// TwinCAT 3 PLC project MasterController
// ProgramVersion: 3.1.4024.0
// libraries:
//   Tc2_EtherCAT, * (Beckhoff Automation GmbH)
//   Tc2_Math, * (Beckhoff Automation GmbH)
//   Tc2_Standard, * (Beckhoff Automation GmbH)
//   Tc2_System, * (Beckhoff Automation GmbH)
//   Tc2_Utilities, * (Beckhoff Automation GmbH)
//   Tc3_Module, * (Beckhoff Automation GmbH)
// project tree:
//   AgiMaths/Frames/ DHTrans.TcPOU (not stored), invFrame.TcPOU (not stored), rotX.TcPOU (not stored), rotY.TcPOU (not stored), rotZ.TcPOU (not stored), transform.TcPOU (not stored)
//   AgiMaths/MatrixLib/ angAxis2Rot.TcPOU (not stored), cross.TcPOU (not stored), Det5.TcPOU (not stored), Det6.TcPOU (not stored), Det7.TcPOU (not stored), invMat6.TcPOU (not stored), invMat6Old.TcPOU (not stored), invMat3.TcPOU (not stored), invMat7.TcPOU (not stored), Mat3T.TcPOU (not stored), matAdd.TcPOU (not stored), matMultiNum.TcPOU (not stored), matMultiply.TcPOU (not stored), matMultiVec.TcPOU (not stored), matSelfAdd.TcPOU (not stored), matSelfSub.TcPOU (not stored), matSub.TcPOU (not stored), matTranspose.TcPOU (not stored), rot2AngAxis.TcPOU (not stored), norm.TcPOU (not stored), normalize.TcPOU (not stored), vecAdd.TcPOU (not stored), vecDot.TcPOU (not stored), vecMultiNum.TcPOU (not stored), vecSelfAdd.TcPOU (not stored), vecSelfMultiNum.TcPOU (not stored), vecSelfSub.TcPOU (not stored), vecSub.TcPOU (not stored)
//   AgiMaths/ sign.TcPOU (not stored), addVec7.TcPOU (not stored), atan2.TcPOU (not stored), cot.TcPOU (not stored)
//   DUTs/Enum/ E_InstruEnergyCtrlWord.TcDUT (not stored), E_InstrumentEnergyType.TcDUT (not stored), E_InstrumentType.TcDUT (not stored), E_MasterArmState.TcDUT (not stored), E_MatchedSlaveArmIdx.TcDUT (not stored), E_SlaveArmState.TcDUT (not stored), E_DriverCtrlWord.TcDUT (not stored), E_DriverOPMode.TcDUT (not stored), E_DriverStatusWord.TcDUT (not stored)
//   DUTs/Structure/MasterSlaveCommunication/ ST_MasterStatus.TcDUT (not stored), ST_SlaveStatus.TcDUT (not stored)
//   DUTs/Structure/ ST_EtherCATState.TcDUT (not stored), ST_InstruStatus.TcDUT (not stored), ST_MatchedMasterArmIdx.TcDUT (not stored), ST_ArmCtrlCmds.TcDUT (not stored), ST_MasterInputDataPool.TcDUT (not stored), ST_Frame.TcDUT (not stored)
//   DUTs/Structure/TasksCommunication/ ST_CartUIData.TcDUT (not stored), ST_MasterDynaData.TcDUT (not stored), ST_MasterUIData.TcDUT (not stored), ST_CartStatus.TcDUT (not stored), ST_MasterJointData.TcDUT (not stored), ST_MotorInputs.TcDUT (not stored), ST_MotorOutputs.TcDUT (not stored), ST_SlaveJointData.TcDUT (not stored), ST_SafetyData.TcDUT (not stored), ST_CartJointData.TcDUT (not stored)
//   DUTs/Structure/UICommunication/ ST_arm_distribution.TcDUT (not stored), ST_ergonCtrlEnable.TcDUT (not stored), ST_ergonomicCtrlData.TcDUT (not stored), ST_instrument_info.TcDUT (not stored), ST_scope_info.TcDUT (not stored)
//   DUTs/Type/ Vec7b.TcDUT (not stored), Mat34.TcDUT (not stored), Mat37.TcDUT (not stored), Mat43.TcDUT (not stored), Mat4d.TcDUT (not stored), Mat5d.TcDUT (not stored), Mat67.TcDUT (not stored), Mat6d.TcDUT (not stored), Mat76.TcDUT (not stored), Mat7d.TcDUT (not stored), Vec4d.TcDUT (not stored), Vec4i.TcDUT (not stored), Vec6i.TcDUT (not stored), Vec4b.TcDUT (not stored), Vec7di.TcDUT (not stored), Vec8d.TcDUT (not stored), Mat3d.TcDUT (not stored), Vec3d.TcDUT (not stored), Vec6d.TcDUT (not stored), Vec7d.TcDUT (not stored), Vec7i.TcDUT (not stored)
//   FBs_Auxiliary/ FB_GripAngleCalc.TcPOU, FB_HandClutchCheck.TcPOU (not stored), FB_IOCheck.TcPOU (not stored), FB_RiseEdgeCheck.TcPOU (not stored), FB_IOToggleCheck.TcPOU (not stored), FB_MSCtrlTriggerCheck.TcPOU (not stored), FB_slaveConnectionCheck.TcPOU (not stored), FB_TON.TcPOU (not stored)
//   FBs_BasicControllers/ FB_boundaryForceFeedback.TcPOU (not stored), FB_Jnt6SWLimit.TcPOU (not stored), FB_PID.TcPOU (not stored), FB_RedunJntControl.TcPOU (not stored)
//   FBs_Observer/ FB_JntObserver.TcPOU (not stored)
//   FBs_RobotDynamics/ FB_MasterDynamic.TcPOU (not stored), FB_MasterFriciton.TcPOU (not stored), FB_MasterGravity.TcPOU (not stored)
//   FBs_Robots/ FB_ArmJoint.TcPOU (not stored), FB_CartJoint.TcPOU, FB_JointBase.TcPOU, FB_MasterCart.TcPOU, FB_MasterArm.TcPOU (not stored), FB_MasterRobot.TcPOU
//   FBs_StateControllers/ FB_EndoscopeController.TcPOU (not stored), FB_StateCtrlClutch.TcPOU (not stored), FB_StateCtrlEndoscope.TcPOU (not stored), FB_StateCtrlCart.TcPOU (not stored), FB_StateCtrlDisable.TcPOU (not stored), FB_StateCtrlGraCali.TcPOU (not stored), FB_StateCtrlMatching.TcPOU, FB_StateCtrlHome.TcPOU (not stored), FB_StateCtrlError.TcPOU (not stored), FB_StateCtrlPerformance.TcPOU (not stored), FB_StateCtrlReady.TcPOU (not stored), FB_StateCtrlMasterSlave.TcPOU (not stored), FB_StateCtrlTest.TcPOU (not stored), FB_StateCtrlInit.TcPOU (not stored), FB_StateCtrlStandBy.TcPOU (not stored), FB_MasterArmCtrlBase.TcPOU (not stored), I_MasterArmCtrl.TcIO (not stored)
//   FBs_TrajectoryPlanning/ FB_BasicDoubleS.TcPOU (not stored), FB_trajBase.TcPOU (not stored), FB_TrajMoveJ.TcPOU (not stored), linear_trajectory_with_quintic_polynomial_blends.TcPOU (not stored), quintic_spline_curve.TcPOU (not stored), Quintic_spline_curve_factor.TcPOU (not stored), TrapezoIDal_velocity_trajectory.TcPOU (not stored)
//   FBs_TrajectoryPlanning/OTG/ FB_secOrdTrajFilter.TcPOU (not stored), FB_thirdOrdTrajFilter.TcPOU (not stored)
//   FBs_Filters/ FB_LowPassFilter.TcPOU (not stored)
//   GVLs/Arms/ GVL_ArmDynamics.TcGVL, GVL_ArmJointCaliData.TcGVL, GVL_ArmKinematic.TcGVL, GVL_ControlParameters.TcGVL (not stored), GVL_ArmJointParameters.TcGVL (not stored)
//   GVLs/Cart/ GVL_CartJointCaliData.TcGVL (not stored), GVL_CartJointParameters.TcGVL (not stored)
//   GVLs/Configs/Robot3/ GVL_ArmDynamics_3.TcGVL (not stored), GVL_ArmJointCaliData_3.TcGVL (not stored), GVL_CartJointCaliData_3.TcGVL (not stored)
//   GVLs/Configs/Robot4/ GVL_ArmDynamics_4.TcGVL (not stored), GVL_ArmJointCaliData_4.TcGVL (not stored), GVL_CartJointCaliData_4_1.TcGVL (not stored)
//   GVLs/Configs/Robot5/ GVL_ArmDynamics_5.TcGVL (not stored), GVL_ArmJointCaliData_5.TcGVL (not stored), GVL_CartJointCaliData_5.TcGVL (not stored)
//   GVLs/Configs/Robot6/ GVL_ArmDynamics_6.TcGVL (not stored), GVL_ArmJointCaliData_6.TcGVL (not stored), GVL_CartJointCaliData_6.TcGVL (not stored)
//   GVLs/ GVL_interactUI.TcGVL (not stored), GVL_MathDefine.TcGVL (not stored), GVL_SafetyParameters.TcGVL, GVL_SystemParameters.TcGVL (not stored)
//   Mains/ CartControl.TcPOU (not stored), SafetyCheck.TcPOU (not stored), MasterArmControl.TcPOU (not stored), RobotDynamics.TcPOU (not stored)
//   SafetyCheck/ ASSERT.TcPOU (not stored), Fb_dataRecord.TcPOU (not stored), FB_EtherCATCheck.TcPOU (not stored), Fb_SafetyCheck.TcPOU, FB_Writer.TcPOU (not stored)
//   SafetyCheck/safetyCheckDUT/ checkDelay.TcDUT (not stored), checkDelayTime.TcDUT (not stored), checkInputVariable.TcDUT (not stored), checkPermit.TcDUT (not stored), ST_Buffer.TcDUT (not stored), T_Buffer.TcDUT (not stored)
//   Sandbox/ FB_CartCheck.TcPOU (not stored), FB_MasterArmCheck.TcPOU (not stored), FB_RedunJntControl_bak2.TcPOU (not stored), FB_RedunJntControl_bak.TcPOU (not stored)
//   / TaskArmControl.TcTTO (not stored), TaskCartControl.TcTTO (not stored), TaskDynamic.TcTTO (not stored), TaskSafetyCheck.TcTTO (not stored)
// real-time tasks:
//   TASK TaskArmControl: cycle T#250us, priority 1, ADS port 350
//   TASK TaskDynamic: cycle T#1ms, priority 2, ADS port 351
//   TASK TaskSafetyCheck: cycle T#1ms, priority 5, ADS port 352
//   TASK TaskCartControl: cycle T#1ms, priority 4, ADS port 353
// I/O:
//   DEVICE RightArm (EtherCAT), AmsNetId 169.254.219.236.5.1
//     Term 7 (EK1100) [EK1100 EtherCAT Coupler (2A E-Bus)]
//       Term 8 (EL6070) [EL6070 1Ch. Licensing-Terminal]
//       Term 9 (EL1008) [EL1008 8Ch. Dig. Input 24V, 3ms]
//       Term 10 (EL1008) [EL1008 8Ch. Dig. Input 24V, 3ms]
//       Term 11 (EL1008) [EL1008 8Ch. Dig. Input 24V, 3ms]
//       Term 12 (EK1122) [EK1122 2 port EtherCAT junction]
//         Box 13 (AX58200_MotorControl) [AX58200_MotorControl_for_1axis]
//         Box 14 (AX58200_MotorControl) [AX58200_MotorControl_for_1axis]
//         Box 15 (AX58200_MotorControl) [AX58200_MotorControl_for_1axis]
//         Box 16 (AX58200_MotorControl) [AX58200_MotorControl_for_1axis]
//     Joint12 [AX58200_MotorControl_Master123]
//     Joint3 [AX58200_MotorControl_Master123]
//     Joint4 [AX58200_MotorControl_for_1axis]
//     Joint5 [AX58200_MotorControl_for_1axis]
//     Joint6 [AX58200_MotorControl_for_1axis]
//     Joint7 [AX58200_MotorControl_for_1axis]
//   DEVICE LeftArm (EtherCAT), AmsNetId 169.254.79.95.2.1
//     Joint12 [AX58200_MotorControl_Master123]
//     Joint3 [AX58200_MotorControl_Master123]
//     Joint4 [AX58200_MotorControl_for_1axis]
//     Joint5 [AX58200_MotorControl_for_1axis]
//     Joint6 [AX58200_MotorControl_for_1axis]
//     Joint7 [AX58200_MotorControl_for_1axis]
//   DEVICE Device 3 (EtherCAT), AmsNetId 169.254.219.236.4.1
//     Box 2 (AX58200_MotorControl) [AX58200_MotorControlHFK]
//     Box 1 (EL6695-0002) [EL6695 EtherCAT Bridge terminal (Secondary)]
// variable links:
//   MasterController/MasterController Instance <-> Device 3 (EtherCAT)/Box 1 (EL6695-0002)
//     TaskArmControl Inputs/MasterArmControl.m_slaveRobotData <-> IO Inputs/SlaveRobotData
//     TaskArmControl Outputs/MasterArmControl.m_masterRobotData <-> IO Outputs/MasterRobotData
//   MasterController/MasterController Instance <-> Device 3 (EtherCAT)/Box 2 (AX58200_MotorControl)
//     TaskCartControl Outputs/CartControl.m_masterCart.m_elecKnifeCtrlWord <-> RxPdoMappingCspCsv/Target velocity
//   MasterController/MasterController Instance <-> LeftArm (EtherCAT)/Joint12
//     TaskArmControl Inputs/MasterArmControl.m_masterRobot.m_masterArms[1].m_joints[1].m_motorInputs/m_current <-> TxPdoMappingCspCsv/Torque actual value
//     TaskArmControl Inputs/MasterArmControl.m_masterRobot.m_masterArms[1].m_joints[1].m_motorInputs/m_driverError <-> TxPdoMappingCspCsv/digital input
//     TaskArmControl Inputs/MasterArmControl.m_masterRobot.m_masterArms[1].m_joints[2].m_motorInputs/m_driverError <-> TxPdoMappingCspCsv/digital input
//     TaskArmControl Inputs/MasterArmControl.m_masterRobot.m_masterArms[1].m_joints[1].m_motorInputs/m_motorEncoder <-> TxPdoMappingCspCsv/Position actual value
//     TaskArmControl Inputs/MasterArmControl.m_masterRobot.m_masterArms[1].m_joints[1].m_motorInputs/m_statusWord <-> TxPdoMappingCspCsv/Statusword
//     TaskArmControl Inputs/MasterArmControl.m_masterRobot.m_masterArms[1].m_joints[2].m_motorInputs/m_statusWord <-> TxPdoMappingCspCsv/Statusword
//     TaskArmControl Inputs/MasterArmControl.m_masterRobot.m_masterArms[1].m_joints[2].m_motorInputs/m_current <-> TxPdoMappingCspCsv/Torque actual value for aix2
//     TaskArmControl Inputs/MasterArmControl.m_masterRobot.m_masterArms[1].m_joints[2].m_motorInputs/m_motorEncoder <-> TxPdoMappingCspCsv/Position actual value for aix2
//     TaskArmControl Inputs/MasterArmControl.m_masterRobot.m_masterArms[1].m_joints[3].m_motorInputs/m_linkEncoder <-> TxPdoMappingCspCsv/ENC2
//     TaskArmControl Outputs/MasterArmControl.m_masterRobot.m_masterArms[1].m_joints[1].m_motorOutputs/m_cmdCurrent <-> RxPdoMappingCspCsv/Target torque
//     TaskArmControl Outputs/MasterArmControl.m_masterRobot.m_masterArms[1].m_joints[1].m_motorOutputs/m_cmdMotorEncoder <-> RxPdoMappingCspCsv/Target position
//     TaskArmControl Outputs/MasterArmControl.m_masterRobot.m_masterArms[1].m_joints[1].m_motorOutputs/m_controlWord <-> RxPdoMappingCspCsv/Controlword
//     TaskArmControl Outputs/MasterArmControl.m_masterRobot.m_masterArms[1].m_joints[1].m_motorOutputs/m_opMode <-> RxPdoMappingCspCsv/Modes of operation
//     TaskArmControl Outputs/MasterArmControl.m_masterRobot.m_masterArms[1].m_joints[2].m_motorOutputs/m_cmdCurrent <-> RxPdoMappingCspCsv/Target Torque value for aix2
//     TaskArmControl Outputs/MasterArmControl.m_masterRobot.m_masterArms[1].m_joints[2].m_motorOutputs/m_cmdMotorEncoder <-> RxPdoMappingCspCsv/Target position value for aix2
//   MasterController/MasterController Instance <-> LeftArm (EtherCAT)/Joint3
//     TaskArmControl Inputs/MasterArmControl.m_masterRobot.m_masterArms[1].m_joints[1].m_motorInputs/m_linkEncoder <-> TxPdoMappingCspCsv/ENC2
//     TaskArmControl Inputs/MasterArmControl.m_masterRobot.m_masterArms[1].m_joints[3].m_motorInputs/m_current <-> TxPdoMappingCspCsv/Torque actual value
//     TaskArmControl Inputs/MasterArmControl.m_masterRobot.m_masterArms[1].m_joints[3].m_motorInputs/m_driverError <-> TxPdoMappingCspCsv/digital input
//     TaskArmControl Inputs/MasterArmControl.m_masterRobot.m_masterArms[1].m_joints[3].m_motorInputs/m_motorEncoder <-> TxPdoMappingCspCsv/Position actual value
//     TaskArmControl Inputs/MasterArmControl.m_masterRobot.m_masterArms[1].m_joints[3].m_motorInputs/m_statusWord <-> TxPdoMappingCspCsv/Statusword
//     TaskArmControl Outputs/MasterArmControl.m_masterRobot.m_masterArms[1].m_joints[3].m_motorOutputs/m_cmdCurrent <-> RxPdoMappingCspCsv/Target torque
//     TaskArmControl Outputs/MasterArmControl.m_masterRobot.m_masterArms[1].m_joints[3].m_motorOutputs/m_cmdMotorEncoder <-> RxPdoMappingCspCsv/Target position
//     TaskArmControl Outputs/MasterArmControl.m_masterRobot.m_masterArms[1].m_joints[3].m_motorOutputs/m_controlWord <-> RxPdoMappingCspCsv/Controlword
//     TaskArmControl Outputs/MasterArmControl.m_masterRobot.m_masterArms[1].m_joints[3].m_motorOutputs/m_opMode <-> RxPdoMappingCspCsv/Modes of operation
//   MasterController/MasterController Instance <-> LeftArm (EtherCAT)/Joint4
//     TaskArmControl Inputs/MasterArmControl.m_masterRobot.m_masterArms[1].m_joints[2].m_motorInputs/m_linkEncoder <-> TxPdoMappingCspCsv/Velocity actual value
//     TaskArmControl Inputs/MasterArmControl.m_masterRobot.m_masterArms[1].m_joints[4].m_motorInputs/m_current <-> TxPdoMappingCspCsv/Torque actual value
//     TaskArmControl Inputs/MasterArmControl.m_masterRobot.m_masterArms[1].m_joints[4].m_motorInputs/m_driverError <-> TxPdoMappingCspCsv/digital input
//     TaskArmControl Inputs/MasterArmControl.m_masterRobot.m_masterArms[1].m_joints[4].m_motorInputs/m_linkEncoder <-> TxPdoMappingCspCsv/ENC2
//     TaskArmControl Inputs/MasterArmControl.m_masterRobot.m_masterArms[1].m_joints[4].m_motorInputs/m_motorEncoder <-> TxPdoMappingCspCsv/Position actual value
//     TaskArmControl Inputs/MasterArmControl.m_masterRobot.m_masterArms[1].m_joints[4].m_motorInputs/m_statusWord <-> TxPdoMappingCspCsv/Statusword
//     TaskArmControl Outputs/MasterArmControl.m_masterRobot.m_masterArms[1].m_joints[4].m_motorOutputs/m_cmdCurrent <-> RxPdoMappingCspCsv/Target torque
//     TaskArmControl Outputs/MasterArmControl.m_masterRobot.m_masterArms[1].m_joints[4].m_motorOutputs/m_cmdMotorEncoder <-> RxPdoMappingCspCsv/Target position
//     TaskArmControl Outputs/MasterArmControl.m_masterRobot.m_masterArms[1].m_joints[4].m_motorOutputs/m_controlWord <-> RxPdoMappingCspCsv/Controlword
//     TaskArmControl Outputs/MasterArmControl.m_masterRobot.m_masterArms[1].m_joints[4].m_motorOutputs/m_opMode <-> RxPdoMappingCspCsv/Modes of operation
//   MasterController/MasterController Instance <-> LeftArm (EtherCAT)/Joint5
//     TaskArmControl Inputs/MasterArmControl.m_masterRobot.m_masterArms[1].m_joints[5].m_motorInputs/m_current <-> TxPdoMappingCspCsv/Torque actual value
//     TaskArmControl Inputs/MasterArmControl.m_masterRobot.m_masterArms[1].m_joints[5].m_motorInputs/m_driverError <-> TxPdoMappingCspCsv/digital input
//     TaskArmControl Inputs/MasterArmControl.m_masterRobot.m_masterArms[1].m_joints[5].m_motorInputs/m_linkEncoder <-> TxPdoMappingCspCsv/ENC2
//     TaskArmControl Inputs/MasterArmControl.m_masterRobot.m_masterArms[1].m_joints[5].m_motorInputs/m_motorEncoder <-> TxPdoMappingCspCsv/Position actual value
//     TaskArmControl Inputs/MasterArmControl.m_masterRobot.m_masterArms[1].m_joints[5].m_motorInputs/m_statusWord <-> TxPdoMappingCspCsv/Statusword
//     TaskArmControl Outputs/MasterArmControl.m_masterRobot.m_masterArms[1].m_joints[5].m_motorOutputs/m_cmdCurrent <-> RxPdoMappingCspCsv/Target torque
//     TaskArmControl Outputs/MasterArmControl.m_masterRobot.m_masterArms[1].m_joints[5].m_motorOutputs/m_cmdMotorEncoder <-> RxPdoMappingCspCsv/Target position
//     TaskArmControl Outputs/MasterArmControl.m_masterRobot.m_masterArms[1].m_joints[5].m_motorOutputs/m_controlWord <-> RxPdoMappingCspCsv/Controlword
//     TaskArmControl Outputs/MasterArmControl.m_masterRobot.m_masterArms[1].m_joints[5].m_motorOutputs/m_opMode <-> RxPdoMappingCspCsv/Modes of operation
//   MasterController/MasterController Instance <-> LeftArm (EtherCAT)/Joint6
//     TaskArmControl Inputs/MasterArmControl.m_masterRobot.m_masterArms[1].m_joints[6].m_motorInputs/m_current <-> TxPdoMappingCspCsv/Torque actual value
//     TaskArmControl Inputs/MasterArmControl.m_masterRobot.m_masterArms[1].m_joints[6].m_motorInputs/m_driverError <-> TxPdoMappingCspCsv/digital input
//     TaskArmControl Inputs/MasterArmControl.m_masterRobot.m_masterArms[1].m_joints[6].m_motorInputs/m_linkEncoder <-> TxPdoMappingCspCsv/ENC2
//     TaskArmControl Inputs/MasterArmControl.m_masterRobot.m_masterArms[1].m_joints[6].m_motorInputs/m_motorEncoder <-> TxPdoMappingCspCsv/Position actual value
//     TaskArmControl Inputs/MasterArmControl.m_masterRobot.m_masterArms[1].m_joints[6].m_motorInputs/m_statusWord <-> TxPdoMappingCspCsv/Statusword
//     TaskArmControl Outputs/MasterArmControl.m_masterRobot.m_masterArms[1].m_joints[6].m_motorOutputs/m_cmdCurrent <-> RxPdoMappingCspCsv/Target torque
//     TaskArmControl Outputs/MasterArmControl.m_masterRobot.m_masterArms[1].m_joints[6].m_motorOutputs/m_cmdMotorEncoder <-> RxPdoMappingCspCsv/Target position
//     TaskArmControl Outputs/MasterArmControl.m_masterRobot.m_masterArms[1].m_joints[6].m_motorOutputs/m_controlWord <-> RxPdoMappingCspCsv/Controlword
//     TaskArmControl Outputs/MasterArmControl.m_masterRobot.m_masterArms[1].m_joints[6].m_motorOutputs/m_opMode <-> RxPdoMappingCspCsv/Modes of operation
//   MasterController/MasterController Instance <-> LeftArm (EtherCAT)/Joint7
//     TaskArmControl Inputs/MasterArmControl.m_masterRobot.m_masterArms[1].m_gripHallSensorIO <-> TxPdoMappingCspCsv/analog input
//     TaskArmControl Inputs/MasterArmControl.m_masterRobot.m_masterArms[1].m_handClutchIO <-> TxPdoMappingCspCsv/digital input
//     TaskArmControl Inputs/MasterArmControl.m_masterRobot.m_masterArms[1].m_joints[7].m_motorInputs/m_current <-> TxPdoMappingCspCsv/Torque actual value
//     TaskArmControl Inputs/MasterArmControl.m_masterRobot.m_masterArms[1].m_joints[7].m_motorInputs/m_linkEncoder <-> TxPdoMappingCspCsv/ENC2
//     TaskArmControl Inputs/MasterArmControl.m_masterRobot.m_masterArms[1].m_joints[7].m_motorInputs/m_motorEncoder <-> TxPdoMappingCspCsv/Position actual value
//     TaskArmControl Inputs/MasterArmControl.m_masterRobot.m_masterArms[1].m_joints[7].m_motorInputs/m_statusWord <-> TxPdoMappingCspCsv/Statusword
//     TaskArmControl Outputs/MasterArmControl.m_masterRobot.m_masterArms[1].m_joints[7].m_motorOutputs/m_cmdCurrent <-> RxPdoMappingCspCsv/Target torque
//     TaskArmControl Outputs/MasterArmControl.m_masterRobot.m_masterArms[1].m_joints[7].m_motorOutputs/m_cmdMotorEncoder <-> RxPdoMappingCspCsv/Target position
//     TaskArmControl Outputs/MasterArmControl.m_masterRobot.m_masterArms[1].m_joints[7].m_motorOutputs/m_controlWord <-> RxPdoMappingCspCsv/Controlword
//     TaskArmControl Outputs/MasterArmControl.m_masterRobot.m_masterArms[1].m_joints[7].m_motorOutputs/m_opMode <-> RxPdoMappingCspCsv/Modes of operation
//   MasterController/MasterController Instance <-> RightArm (EtherCAT)/Joint12
//     TaskArmControl Inputs/MasterArmControl.m_masterRobot.m_masterArms[2].m_joints[1].m_motorInputs/m_current <-> TxPdoMappingCspCsv/Torque actual value
//     TaskArmControl Inputs/MasterArmControl.m_masterRobot.m_masterArms[2].m_joints[1].m_motorInputs/m_driverError <-> TxPdoMappingCspCsv/digital input
//     TaskArmControl Inputs/MasterArmControl.m_masterRobot.m_masterArms[2].m_joints[1].m_motorInputs/m_motorEncoder <-> TxPdoMappingCspCsv/Position actual value
//     TaskArmControl Inputs/MasterArmControl.m_masterRobot.m_masterArms[2].m_joints[1].m_motorInputs/m_statusWord <-> TxPdoMappingCspCsv/Statusword
//     TaskArmControl Inputs/MasterArmControl.m_masterRobot.m_masterArms[2].m_joints[2].m_motorInputs/m_statusWord <-> TxPdoMappingCspCsv/Statusword
//     TaskArmControl Inputs/MasterArmControl.m_masterRobot.m_masterArms[2].m_joints[2].m_motorInputs/m_current <-> TxPdoMappingCspCsv/Torque actual value for aix2
//     TaskArmControl Inputs/MasterArmControl.m_masterRobot.m_masterArms[2].m_joints[2].m_motorInputs/m_motorEncoder <-> TxPdoMappingCspCsv/Position actual value for aix2
//     TaskArmControl Inputs/MasterArmControl.m_masterRobot.m_masterArms[2].m_joints[3].m_motorInputs/m_linkEncoder <-> TxPdoMappingCspCsv/ENC2
//     TaskArmControl Outputs/MasterArmControl.m_masterRobot.m_masterArms[2].m_joints[1].m_motorOutputs/m_cmdCurrent <-> RxPdoMappingCspCsv/Target torque
//     TaskArmControl Outputs/MasterArmControl.m_masterRobot.m_masterArms[2].m_joints[1].m_motorOutputs/m_cmdMotorEncoder <-> RxPdoMappingCspCsv/Target position
//     TaskArmControl Outputs/MasterArmControl.m_masterRobot.m_masterArms[2].m_joints[1].m_motorOutputs/m_controlWord <-> RxPdoMappingCspCsv/Controlword
//     TaskArmControl Outputs/MasterArmControl.m_masterRobot.m_masterArms[2].m_joints[1].m_motorOutputs/m_opMode <-> RxPdoMappingCspCsv/Modes of operation
//     TaskArmControl Outputs/MasterArmControl.m_masterRobot.m_masterArms[2].m_joints[2].m_motorOutputs/m_cmdCurrent <-> RxPdoMappingCspCsv/Target Torque value for aix2
//     TaskArmControl Outputs/MasterArmControl.m_masterRobot.m_masterArms[2].m_joints[2].m_motorOutputs/m_cmdMotorEncoder <-> RxPdoMappingCspCsv/Target position value for aix2
//   MasterController/MasterController Instance <-> RightArm (EtherCAT)/Joint3
//     TaskArmControl Inputs/MasterArmControl.m_masterRobot.m_masterArms[2].m_joints[1].m_motorInputs/m_linkEncoder <-> TxPdoMappingCspCsv/ENC2
//     TaskArmControl Inputs/MasterArmControl.m_masterRobot.m_masterArms[2].m_joints[3].m_motorInputs/m_current <-> TxPdoMappingCspCsv/Torque actual value
//     TaskArmControl Inputs/MasterArmControl.m_masterRobot.m_masterArms[2].m_joints[3].m_motorInputs/m_driverError <-> TxPdoMappingCspCsv/digital input
//     TaskArmControl Inputs/MasterArmControl.m_masterRobot.m_masterArms[2].m_joints[3].m_motorInputs/m_motorEncoder <-> TxPdoMappingCspCsv/Position actual value
//     TaskArmControl Inputs/MasterArmControl.m_masterRobot.m_masterArms[2].m_joints[3].m_motorInputs/m_statusWord <-> TxPdoMappingCspCsv/Statusword
//     TaskArmControl Outputs/MasterArmControl.m_masterRobot.m_masterArms[2].m_joints[3].m_motorOutputs/m_cmdCurrent <-> RxPdoMappingCspCsv/Target torque
//     TaskArmControl Outputs/MasterArmControl.m_masterRobot.m_masterArms[2].m_joints[3].m_motorOutputs/m_cmdMotorEncoder <-> RxPdoMappingCspCsv/Target position
//     TaskArmControl Outputs/MasterArmControl.m_masterRobot.m_masterArms[2].m_joints[3].m_motorOutputs/m_controlWord <-> RxPdoMappingCspCsv/Controlword
//     TaskArmControl Outputs/MasterArmControl.m_masterRobot.m_masterArms[2].m_joints[3].m_motorOutputs/m_opMode <-> RxPdoMappingCspCsv/Modes of operation
//   MasterController/MasterController Instance <-> RightArm (EtherCAT)/Joint4
//     TaskArmControl Inputs/MasterArmControl.m_masterRobot.m_masterArms[2].m_joints[2].m_motorInputs/m_linkEncoder <-> TxPdoMappingCspCsv/Velocity actual value
//     TaskArmControl Inputs/MasterArmControl.m_masterRobot.m_masterArms[2].m_joints[4].m_motorInputs/m_current <-> TxPdoMappingCspCsv/Torque actual value
//     TaskArmControl Inputs/MasterArmControl.m_masterRobot.m_masterArms[2].m_joints[4].m_motorInputs/m_driverError <-> TxPdoMappingCspCsv/digital input
//     TaskArmControl Inputs/MasterArmControl.m_masterRobot.m_masterArms[2].m_joints[4].m_motorInputs/m_linkEncoder <-> TxPdoMappingCspCsv/ENC2
//     TaskArmControl Inputs/MasterArmControl.m_masterRobot.m_masterArms[2].m_joints[4].m_motorInputs/m_motorEncoder <-> TxPdoMappingCspCsv/Position actual value
//     TaskArmControl Inputs/MasterArmControl.m_masterRobot.m_masterArms[2].m_joints[4].m_motorInputs/m_statusWord <-> TxPdoMappingCspCsv/Statusword
//     TaskArmControl Outputs/MasterArmControl.m_masterRobot.m_masterArms[2].m_joints[4].m_motorOutputs/m_cmdCurrent <-> RxPdoMappingCspCsv/Target torque
//     TaskArmControl Outputs/MasterArmControl.m_masterRobot.m_masterArms[2].m_joints[4].m_motorOutputs/m_cmdMotorEncoder <-> RxPdoMappingCspCsv/Target position
//     TaskArmControl Outputs/MasterArmControl.m_masterRobot.m_masterArms[2].m_joints[4].m_motorOutputs/m_controlWord <-> RxPdoMappingCspCsv/Controlword
//     TaskArmControl Outputs/MasterArmControl.m_masterRobot.m_masterArms[2].m_joints[4].m_motorOutputs/m_opMode <-> RxPdoMappingCspCsv/Modes of operation
//   MasterController/MasterController Instance <-> RightArm (EtherCAT)/Joint5
//     TaskArmControl Inputs/MasterArmControl.m_masterRobot.m_masterArms[2].m_joints[5].m_motorInputs/m_current <-> TxPdoMappingCspCsv/Torque actual value
//     TaskArmControl Inputs/MasterArmControl.m_masterRobot.m_masterArms[2].m_joints[5].m_motorInputs/m_driverError <-> TxPdoMappingCspCsv/digital input
//     TaskArmControl Inputs/MasterArmControl.m_masterRobot.m_masterArms[2].m_joints[5].m_motorInputs/m_linkEncoder <-> TxPdoMappingCspCsv/ENC2
//     TaskArmControl Inputs/MasterArmControl.m_masterRobot.m_masterArms[2].m_joints[5].m_motorInputs/m_motorEncoder <-> TxPdoMappingCspCsv/Position actual value
//     TaskArmControl Inputs/MasterArmControl.m_masterRobot.m_masterArms[2].m_joints[5].m_motorInputs/m_statusWord <-> TxPdoMappingCspCsv/Statusword
//     TaskArmControl Outputs/MasterArmControl.m_masterRobot.m_masterArms[2].m_joints[5].m_motorOutputs/m_cmdCurrent <-> RxPdoMappingCspCsv/Target torque
//     TaskArmControl Outputs/MasterArmControl.m_masterRobot.m_masterArms[2].m_joints[5].m_motorOutputs/m_cmdMotorEncoder <-> RxPdoMappingCspCsv/Target position
//     TaskArmControl Outputs/MasterArmControl.m_masterRobot.m_masterArms[2].m_joints[5].m_motorOutputs/m_controlWord <-> RxPdoMappingCspCsv/Controlword
//     TaskArmControl Outputs/MasterArmControl.m_masterRobot.m_masterArms[2].m_joints[5].m_motorOutputs/m_opMode <-> RxPdoMappingCspCsv/Modes of operation
//   MasterController/MasterController Instance <-> RightArm (EtherCAT)/Joint6
//     TaskArmControl Inputs/MasterArmControl.m_masterRobot.m_masterArms[2].m_joints[6].m_motorInputs/m_current <-> TxPdoMappingCspCsv/Torque actual value
//     TaskArmControl Inputs/MasterArmControl.m_masterRobot.m_masterArms[2].m_joints[6].m_motorInputs/m_driverError <-> TxPdoMappingCspCsv/digital input
//     TaskArmControl Inputs/MasterArmControl.m_masterRobot.m_masterArms[2].m_joints[6].m_motorInputs/m_linkEncoder <-> TxPdoMappingCspCsv/ENC2
//     TaskArmControl Inputs/MasterArmControl.m_masterRobot.m_masterArms[2].m_joints[6].m_motorInputs/m_motorEncoder <-> TxPdoMappingCspCsv/Position actual value
//     TaskArmControl Inputs/MasterArmControl.m_masterRobot.m_masterArms[2].m_joints[6].m_motorInputs/m_statusWord <-> TxPdoMappingCspCsv/Statusword
//     TaskArmControl Outputs/MasterArmControl.m_masterRobot.m_masterArms[2].m_joints[6].m_motorOutputs/m_cmdCurrent <-> RxPdoMappingCspCsv/Target torque
//     TaskArmControl Outputs/MasterArmControl.m_masterRobot.m_masterArms[2].m_joints[6].m_motorOutputs/m_cmdMotorEncoder <-> RxPdoMappingCspCsv/Target position
//     TaskArmControl Outputs/MasterArmControl.m_masterRobot.m_masterArms[2].m_joints[6].m_motorOutputs/m_controlWord <-> RxPdoMappingCspCsv/Controlword
//     TaskArmControl Outputs/MasterArmControl.m_masterRobot.m_masterArms[2].m_joints[6].m_motorOutputs/m_opMode <-> RxPdoMappingCspCsv/Modes of operation
//   MasterController/MasterController Instance <-> RightArm (EtherCAT)/Joint7
//     TaskArmControl Inputs/MasterArmControl.m_masterRobot.m_masterArms[2].m_gripHallSensorIO <-> TxPdoMappingCspCsv/analog input
//     TaskArmControl Inputs/MasterArmControl.m_masterRobot.m_masterArms[2].m_handClutchIO <-> TxPdoMappingCspCsv/digital input
//     TaskArmControl Inputs/MasterArmControl.m_masterRobot.m_masterArms[2].m_joints[7].m_motorInputs/m_current <-> TxPdoMappingCspCsv/Torque actual value
//     TaskArmControl Inputs/MasterArmControl.m_masterRobot.m_masterArms[2].m_joints[7].m_motorInputs/m_linkEncoder <-> TxPdoMappingCspCsv/ENC2
//     TaskArmControl Inputs/MasterArmControl.m_masterRobot.m_masterArms[2].m_joints[7].m_motorInputs/m_motorEncoder <-> TxPdoMappingCspCsv/Position actual value
//     TaskArmControl Inputs/MasterArmControl.m_masterRobot.m_masterArms[2].m_joints[7].m_motorInputs/m_statusWord <-> TxPdoMappingCspCsv/Statusword
//     TaskArmControl Outputs/MasterArmControl.m_masterRobot.m_masterArms[2].m_joints[7].m_motorOutputs/m_cmdCurrent <-> RxPdoMappingCspCsv/Target torque
//     TaskArmControl Outputs/MasterArmControl.m_masterRobot.m_masterArms[2].m_joints[7].m_motorOutputs/m_cmdMotorEncoder <-> RxPdoMappingCspCsv/Target position
//     TaskArmControl Outputs/MasterArmControl.m_masterRobot.m_masterArms[2].m_joints[7].m_motorOutputs/m_controlWord <-> RxPdoMappingCspCsv/Controlword
//     TaskArmControl Outputs/MasterArmControl.m_masterRobot.m_masterArms[2].m_joints[7].m_motorOutputs/m_opMode <-> RxPdoMappingCspCsv/Modes of operation
//   MasterController/MasterController Instance <-> RightArm (EtherCAT)/Term 7 (EK1100)/Term 10 (EL1008)
//     TaskCartControl Inputs/CartControl.m_masterCart.m_electricCoagulLeftAllow <-> Channel 2/electricCoagulLeftAllow
//     TaskCartControl Inputs/CartControl.m_masterCart.m_electricCoagulRightAllow <-> Channel 4/electricCoagulRightAllow
//     TaskCartControl Inputs/CartControl.m_masterCart.m_electricCutLeftAllow <-> Channel 1/electricCutlLeftAllow
//     TaskCartControl Inputs/CartControl.m_masterCart.m_electricCutRightAllow <-> Channel 3/electricCutRightAllow
//     TaskCartControl Inputs/CartControl.m_masterCart.m_surgonHeadInIO <-> Channel 5/surgonHeadIn
//     TaskSafetyCheck Inputs/SafetyCheck.m_cartLockSignalLeft <-> Channel 7/CartLockSignalLeft
//     TaskSafetyCheck Inputs/SafetyCheck.m_cartLockSignalRight <-> Channel 8/CartLockSignalRight
//   MasterController/MasterController Instance <-> RightArm (EtherCAT)/Term 7 (EK1100)/Term 11 (EL1008)
//     TaskCartControl Inputs/CartControl.m_masterCart.m_cartJointCtrlIO[1] <-> Channel 1/Input
//     TaskCartControl Inputs/CartControl.m_masterCart.m_cartJointCtrlIO[2] <-> Channel 2/Input
//     TaskCartControl Inputs/CartControl.m_masterCart.m_cartJointCtrlIO[3] <-> Channel 8/Input
//     TaskCartControl Inputs/CartControl.m_masterCart.m_cartJointCtrlIO[4] <-> Channel 7/Input
//     TaskCartControl Inputs/CartControl.m_masterCart.m_cartJointCtrlIO[5] <-> Channel 3/Input
//     TaskCartControl Inputs/CartControl.m_masterCart.m_cartJointCtrlIO[6] <-> Channel 4/Input
//     TaskCartControl Inputs/CartControl.m_masterCart.m_cartJointCtrlIO[7] <-> Channel 6/Input
//     TaskCartControl Inputs/CartControl.m_masterCart.m_cartJointCtrlIO[8] <-> Channel 5/Input
//   MasterController/MasterController Instance <-> RightArm (EtherCAT)/Term 7 (EK1100)/Term 12 (EK1122)/Box 13 (AX58200_MotorControl)
//     TaskCartControl Inputs/CartControl.m_masterCart.m_cartJoints[3].m_motorInputs/m_current <-> TxPdoMappingCspCsv/Torque actual value
//     TaskCartControl Inputs/CartControl.m_masterCart.m_cartJoints[3].m_motorInputs/m_driverError <-> TxPdoMappingCspCsv/digital input
//     TaskCartControl Inputs/CartControl.m_masterCart.m_cartJoints[3].m_motorInputs/m_linkEncoder <-> TxPdoMappingCspCsv/ENC2
//     TaskCartControl Inputs/CartControl.m_masterCart.m_cartJoints[3].m_motorInputs/m_motorEncoder <-> TxPdoMappingCspCsv/Position actual value
//     TaskCartControl Inputs/CartControl.m_masterCart.m_cartJoints[3].m_motorInputs/m_statusWord <-> TxPdoMappingCspCsv/Statusword
//     TaskCartControl Outputs/CartControl.m_masterCart.m_cartJoints[3].m_motorOutputs/m_cmdCurrent <-> RxPdoMappingCspCsv/Target torque
//     TaskCartControl Outputs/CartControl.m_masterCart.m_cartJoints[3].m_motorOutputs/m_cmdMotorEncoder <-> RxPdoMappingCspCsv/Target position
//     TaskCartControl Outputs/CartControl.m_masterCart.m_cartJoints[3].m_motorOutputs/m_controlWord <-> RxPdoMappingCspCsv/Controlword
//     TaskCartControl Outputs/CartControl.m_masterCart.m_cartJoints[3].m_motorOutputs/m_opMode <-> RxPdoMappingCspCsv/Modes of operation
//   MasterController/MasterController Instance <-> RightArm (EtherCAT)/Term 7 (EK1100)/Term 12 (EK1122)/Box 14 (AX58200_MotorControl)
//     TaskCartControl Inputs/CartControl.m_masterCart.m_cartJoints[1].m_motorInputs/m_current <-> TxPdoMappingCspCsv/Torque actual value
//     TaskCartControl Inputs/CartControl.m_masterCart.m_cartJoints[1].m_motorInputs/m_driverError <-> TxPdoMappingCspCsv/digital input
//     TaskCartControl Inputs/CartControl.m_masterCart.m_cartJoints[1].m_motorInputs/m_linkEncoder <-> TxPdoMappingCspCsv/ENC2
//     TaskCartControl Inputs/CartControl.m_masterCart.m_cartJoints[1].m_motorInputs/m_motorEncoder <-> TxPdoMappingCspCsv/Position actual value
//     TaskCartControl Inputs/CartControl.m_masterCart.m_cartJoints[1].m_motorInputs/m_statusWord <-> TxPdoMappingCspCsv/Statusword
//     TaskCartControl Outputs/CartControl.m_masterCart.m_cartJoints[1].m_motorOutputs/m_cmdCurrent <-> RxPdoMappingCspCsv/Target torque
//     TaskCartControl Outputs/CartControl.m_masterCart.m_cartJoints[1].m_motorOutputs/m_cmdMotorEncoder <-> RxPdoMappingCspCsv/Target position
//     TaskCartControl Outputs/CartControl.m_masterCart.m_cartJoints[1].m_motorOutputs/m_controlWord <-> RxPdoMappingCspCsv/Controlword
//     TaskCartControl Outputs/CartControl.m_masterCart.m_cartJoints[1].m_motorOutputs/m_opMode <-> RxPdoMappingCspCsv/Modes of operation
//   MasterController/MasterController Instance <-> RightArm (EtherCAT)/Term 7 (EK1100)/Term 12 (EK1122)/Box 15 (AX58200_MotorControl)
//     TaskCartControl Inputs/CartControl.m_masterCart.m_cartJoints[4].m_motorInputs/m_current <-> TxPdoMappingCspCsv/Torque actual value
//     TaskCartControl Inputs/CartControl.m_masterCart.m_cartJoints[4].m_motorInputs/m_driverError <-> TxPdoMappingCspCsv/digital input
//     TaskCartControl Inputs/CartControl.m_masterCart.m_cartJoints[4].m_motorInputs/m_linkEncoder <-> TxPdoMappingCspCsv/ENC2
//     TaskCartControl Inputs/CartControl.m_masterCart.m_cartJoints[4].m_motorInputs/m_motorEncoder <-> TxPdoMappingCspCsv/Position actual value
//     TaskCartControl Inputs/CartControl.m_masterCart.m_cartJoints[4].m_motorInputs/m_statusWord <-> TxPdoMappingCspCsv/Statusword
//     TaskCartControl Outputs/CartControl.m_masterCart.m_cartJoints[4].m_motorOutputs/m_cmdCurrent <-> RxPdoMappingCspCsv/Target torque
//     TaskCartControl Outputs/CartControl.m_masterCart.m_cartJoints[4].m_motorOutputs/m_cmdMotorEncoder <-> RxPdoMappingCspCsv/Target position
//     TaskCartControl Outputs/CartControl.m_masterCart.m_cartJoints[4].m_motorOutputs/m_controlWord <-> RxPdoMappingCspCsv/Controlword
//     TaskCartControl Outputs/CartControl.m_masterCart.m_cartJoints[4].m_motorOutputs/m_opMode <-> RxPdoMappingCspCsv/Modes of operation
//   MasterController/MasterController Instance <-> RightArm (EtherCAT)/Term 7 (EK1100)/Term 12 (EK1122)/Box 16 (AX58200_MotorControl)
//     TaskCartControl Inputs/CartControl.m_masterCart.m_cartJoints[2].m_motorInputs/m_current <-> TxPdoMappingCspCsv/Torque actual value
//     TaskCartControl Inputs/CartControl.m_masterCart.m_cartJoints[2].m_motorInputs/m_driverError <-> TxPdoMappingCspCsv/digital input
//     TaskCartControl Inputs/CartControl.m_masterCart.m_cartJoints[2].m_motorInputs/m_linkEncoder <-> TxPdoMappingCspCsv/ENC2
//     TaskCartControl Inputs/CartControl.m_masterCart.m_cartJoints[2].m_motorInputs/m_motorEncoder <-> TxPdoMappingCspCsv/Position actual value
//     TaskCartControl Inputs/CartControl.m_masterCart.m_cartJoints[2].m_motorInputs/m_statusWord <-> TxPdoMappingCspCsv/Statusword
//     TaskCartControl Outputs/CartControl.m_masterCart.m_cartJoints[2].m_motorOutputs/m_cmdCurrent <-> RxPdoMappingCspCsv/Target torque
//     TaskCartControl Outputs/CartControl.m_masterCart.m_cartJoints[2].m_motorOutputs/m_cmdMotorEncoder <-> RxPdoMappingCspCsv/Target position
//     TaskCartControl Outputs/CartControl.m_masterCart.m_cartJoints[2].m_motorOutputs/m_controlWord <-> RxPdoMappingCspCsv/Controlword
//     TaskCartControl Outputs/CartControl.m_masterCart.m_cartJoints[2].m_motorOutputs/m_opMode <-> RxPdoMappingCspCsv/Modes of operation
//   MasterController/MasterController Instance <-> RightArm (EtherCAT)/Term 7 (EK1100)/Term 9 (EL1008)
//     TaskArmControl Inputs/SafetyCheck.m_stopButton <-> Channel 1/StopButton
//     TaskCartControl Inputs/CartControl.m_masterCart.m_armSwitchIO <-> Channel 4/armSwitchIO
//     TaskCartControl Inputs/CartControl.m_masterCart.m_clutchPedalIO <-> Channel 2/clutchPedalIO
//     TaskCartControl Inputs/CartControl.m_masterCart.m_electricCoagulLeft <-> Channel 7/electricCoagulLeft
//     TaskCartControl Inputs/CartControl.m_masterCart.m_electricCoagulRight <-> Channel 8/electricCoagulRight
//     TaskCartControl Inputs/CartControl.m_masterCart.m_electricCutLeft <-> Channel 5/electricCutLeft
//     TaskCartControl Inputs/CartControl.m_masterCart.m_electricCutRight <-> Channel 6/electricCutRight
//     TaskCartControl Inputs/CartControl.m_masterCart.m_endoScopePedalIO <-> Channel 3/endoScopePedaoIO
//   MasterController/MasterController Instance <-> MasterController/MasterController Instance
//     TaskArmControl Inputs/MasterArmControl.m_masterInputDataPool.m_cartStatus <-> TaskCartControl Outputs/CartControl.m_cartStatus
//     TaskArmControl Inputs/MasterArmControl.m_masterInputDataPool.m_masterDynaData <-> TaskDynamic Outputs/RobotDynamics.m_masterDynaData
//     TaskArmControl Inputs/MasterArmControl.m_masterInputDataPool.m_safetyData <-> TaskCartControl Outputs/SafetyCheck.m_safetyCheckData
//     TaskDynamic Inputs/RobotDynamics.m_masterJointsData <-> TaskArmControl Outputs/MasterArmControl.m_masterJointsData
//     TaskSafetyCheck Inputs/SafetyCheck.m_cartJointData <-> TaskCartControl Outputs/CartControl.m_cartJointData
//     TaskSafetyCheck Inputs/SafetyCheck.m_cartStatus <-> TaskCartControl Outputs/CartControl.m_cartStatus
//     TaskSafetyCheck Inputs/SafetyCheck.m_masterJointData <-> TaskArmControl Outputs/MasterArmControl.m_masterJointsData
//     TaskSafetyCheck Inputs/SafetyCheck.m_masterStatus <-> TaskArmControl Outputs/MasterArmControl.m_masterStatus

// ---- GVLs/Arms/GVL_ArmDynamics.TcGVL
{attribute 'global_init_slot' := '49992'}
{attribute 'qualified_only'}
// Robot3 Data
VAR_GLOBAL CONSTANT
	// arm gravity parameters
	(*graParam=[ 2.7244*m3 + 2.7244*m4 + 2.7244*m5 + 2.7244*m6 + 9.8*mx2 + 9.8*mx9,
				9.8*my2 + 9.8*my9,
				3.577*m4 + 3.577*m5 + 3.577*m6 + 0.49*m9 + 9.8*mx3 + 9.8*mx8
				1.5827*m4 + 1.5827*m5 + 1.5827*m6 + 9.8*my3 + 9.8*my8 + 9.8*mz4
				mz5-my4,	my5+mz6,  	mx4,   	mx5, 	mx6,   	my6
				preF2,   k2,   preF3,    k3,    preF5   k5]*)
	g_gravityParam :ARRAY[1..2, 1..16] OF REAL := 
		  [ 5.4276111, -0.0006276305, 3.7625262, 0.86432075, -0.035201665, 0.020692866, 0.000012500212, 0.000035099996, -0.000025502281, -0.012451749, 
			14.60101, 2199.9398, 16.630378, 2907.9775, 4.0032, 756.0, 
		   4.6562429, -0.00071551426, 3.4250331, 0.88315136, -0.037016743, 0.022335894, 0.000037499999, 0.0000117, 0.00026894044, -0.012891512, 
			16.121924, 1920.3613, 7.018418, 2911.5084, 4.0032, 756.0];
			
	// gravity deviation
	g_gravityDeviaion :ARRAY[1..2, 1..7] OF REAL :=
	[ 0.0, 0.0, 0.0, 0.0, -0.00, 0.0, 0.0, 
	 0.0, 0.0, 0.0, 0.0, 0.00, 0.0, 0.0];
	  
	// arm friction parameters [a1,b1,...a7,b7];
	// friction = a * gravity + b; only joint 5 and 6 is identified
	g_jntFrictionParam :ARRAY[1..2, 1..14] OF LREAL :=
	[ 0, 0.058572897, 0.018430306, 0.10524436, -0.0049154602, 0.084832402, 0.31058466, 0.02028806, 0.44112771, 0.0059655609, 0.37723647, 0.0067686593, 0, 0.0028099796,
	 0, 0.058889711, -0.035612353, 0.091429753, 0.034417718, 0.076475174, 0.29029823, 0.030368122, 0.35668967, 0.0072322909, 0.36459748, 0.0077003893, 0, 0.0026510809];
	g_maxJntFriction : Vec7d :=[0.2, 0.2, 0.2, 0.1, 0.1, 0.1, 0.01];
	
	//################ dynamic reference model parameters below ###########################
	// link mass [m1, m2, m3, m4, m5, m6, m7, m8, m9]
	g_linkMass :ARRAY[1..9] OF LREAL :=[2.676, 0.825, 0.547, 0.25, 0.195, 0.194, 0.05, 0.111, 0.09] ;
	
	// lin center of amss
	g_linkCOM :ARRAY[1..9,1..3] OF LREAL := [   1.376E-3,    -1.019E-3,  -81.464E-3,
										   90.622E-3,   -0.113E-3,  15.088E-3,
										   167.4E-3,    3.7E-3,     -0.438E-3,
										   0.1E-3,      98.49E-3,   -55.74E-3,
										   0.12E-3,     76.667E-3,  -36E-3,
										   0,           -61.63E-3,  27.3E-3,
										   0.06E-3,     -0.08E-3,   17.671E-3,
										   11E-3,       -3.364E-3,  39.265E-3,
										   143e-3,      0.495e-3,   24.253e-3];
	// link  inertial
    // [Ixx,Iyy,Izz, Ixy,Ixz, Iyz]
 	g_linkInertia :ARRAY[1..9,1..6] OF LREAL :=[  19.63E-3,   16.43E-3,  12.7E-3,   -0.3222E-3,    -0.667E-3,     -0.0268E-3,
												   1.017E-3,   6.637E-3,  5.935E-3,  -0.037E-3,     -0.238E-3,     0.06E-3,
												   0.161E-3,   9.572E-3,  9.586E-3,  0.0447E-3,     0.0277E-3,     0.465E-6,
												   0.992E-3,   0.707E-3,  0.335E-3,  0.2E-6,     2E-6,       0.224E-3,
												   0.402E-3,   0.25E-3,   0.186E-3,  0.002E-6,   -1.2E-6,    0.106E-3,
												   0.281E-3,   0.178E-3,  0.137E-3,  0.076E-6,   0.09E-6,    0.056E-3,
												   0.0255E-3,  0.0259E-3, 5.96E-6,0.34E-6,    -3E-9,      24E-9,
												   0.033E-3,   0.0976E-3, 0.126E-3,  3E-6,       -5E-6,      -0.162E-6,
												   4.9E-6,  0.757E-3,  0.760E-3,  2.6E-6,     -5.3E-6,    -18E-9];

	//################ DO NOT modify parameters below ###########################
	//  motor inertial at link size
	g_motorInertia :ARRAY[1..7] OF LREAL := [34.7E-7, 34.7E-7, 34.7E-7, 9.26E-7, 0.495E-7, 0.495E-7, 0.495E-7];
	
	// spring parameters
	// spring2 [L0, b1, b2, l1, r0]
	g_spring2Param :ARRAY[1..5] OF LREAL :=[114.3E-3, 20E-3, 16E-3, 200E-3, 30E-3];
	// spring3 [L0, b1, b2, l1, r0,d]
	g_spring3Param :ARRAY[1..6] OF LREAL :=[127.5E-3, 20E-3, 23E-3, 200E-3, 32E-3, 23E-3];
	// spring5 [L0, s1, L1, r0, beta]
	g_spring5Param :ARRAY[1..5] OF LREAL :=[70E-3, 17E-3, 121E-3, 7.5E-3, 32.02*g_deg2rad];
	
END_VAR

// ---- GVLs/Arms/GVL_ArmJointCaliData.TcGVL
{attribute 'qualified_only'}
// Robot3 Data-RightArm
VAR_GLOBAL CONSTANT									 
	// absolute encoder value at minimal joint positon
	g_minLinkEncoder :ARRAY[1..g_mArmNum, 1..g_mJntNum] OF DINT :=
		[122745, 128228, 36292, 22430, 20158, 45700, 0,
		 35855, 68924, 4429, 107164, 130111, 42645, 0];
		 
	// absolute encoder value at maximum joint positon
	g_maxLinkEncoder :ARRAY[1..g_mArmNum, 1..g_mJntNum] OF DINT :=
		[36223, 83720, 69818, 109643, 52927, 65855, 0,
		 79841, 24455, 37956, 63571, 31889, 22283, 0];
	
	// absolute encoder value at calibrated positon
	g_caliLinkEncoder :ARRAY[1..g_mArmNum, 1..g_mJntNum] OF DINT :=
		[15150, 107027, 47903, 76302, 102239, 88760, 53627,
		 57523, 46542, 15769, 8255, 81176, 131007, 56205];
	
	 // if absolute encoder value cross zeros within joint motion range
	 // NOTICE: joint 7 is always 0.
	g_linkEncZeroCross :ARRAY[1..g_mArmNum, 1..g_mJntNum] OF INT :=
		[1, 0, 0, 0, 1, 1, 1,
		 0, 0, 1, 1, 0, 1, 1];
		 
	// limit value of gripper hall sensor
	g_minHallSensorValue :ARRAY[1..2] OF DINT:=[8720383,8982527];
	g_maxHallSensorValue :ARRAY[1..2] OF DINT  :=[95684892,94374153];
		 
 	//################ DO NOT modify parameters below ###########################	
	// abolute encoder expanded limit buffer in case there is calibrtion error at limit position
	g_linkEncLimitBuffer : DINT := 1000;
	
	// flag if joint can rotate multiple cycles
	g_multipleCyclesJoint :ARRAY[1..g_mArmNum, 1..g_mJntNum] OF INT :=
		[0, 0, 0, 0, 0, 0, 1,
		 0, 0, 0, 0, 0, 0, 1];
		 
	// joint position at link encoder calibrated point
	g_linkEncCaliJntPos :ARRAY[1..g_mArmNum, 1..g_mJntNum] OF LREAL :=
		[0.0, -PI/2, 0.0, -pi, pi, -PI/2, 0.0,
		 0.0, -PI/2, 0.0, 0.0, pi, PI/2, 0.0];

END_VAR

// ---- GVLs/Arms/GVL_ArmKinematic.TcGVL
// use slot attribute larger than 49990, which is the default one, if it depends on variable in other file
{attribute 'global_init_slot' := '49991'} 
VAR_GLOBAL CONSTANT 

// distance between shoulders of left and right arm
g_shoulderDistance :LREAL := 0.5;

// master arm shoulder rotation in base monitor pose(0 rotate angle)
g_shoulderRotInMonitor : Mat3d :=[0.0,	-1.0,	0.0,
								  0.0,	0.0,	1.0,
								  -1.0,	0.0,	0.0];
 	
(* 
% DH definetion
% !!!!NOTE: q4 is the DH joint position, NOT the motor one
% paramters definiton:
% d1: arm origin to joint1 
% a3: upper arm length
% a4: lower arm length
% d4: wrist height
% a9: parallel structure width
% DH definition:
% index     parent  alpha   a       theta   d       active
% 1         0       0       0       q1      d1      1
% 2         1       -90     0       q2      0       1
% 3         0       0       a3      q3      0       0
% 4         3       -90     a4      q4      d4      1
% 5         4       90      0       q5      0       1
% 6         5       -90     0       q6      0       1
% 7         6       90      0       q7      0       1

% 8         1       -90     0       q8      0       1
% 9         8       0       a9      q9      0       0
% 10        9       0       a3      q10     0       0
% 11        3       0       a9      0       0       fixed

%q4 = motor_q4+q8-q2-90
%q3 = q8 - q2;
%q9 = q2-q8;
%q10 = q8-q2

*)
g_d1:LREAL:=0.26085;
g_d4:LREAL:=0.156;
g_a3:LREAL:=0.278;
g_a4:LREAL:=0.365;
g_a9:LREAL:=0.06;

//alpha,a,d,theta	
g_masterArmDH:ARRAY[1..9,1..4] OF LREAL :=[0,	0,		g_d1,	0,      
										-pi/2,	0,		0,		0,
										0,		g_a3,	0,		0,
										-pi/2,	g_a4,	g_d4,	0,       
										pi/2,	0,		0,		0,
										-pi/2,	0,		0,		0,
										pi/2,	0,		0,		0,
										-pi/2,	0,		0,		0,// joint 8
										0,		g_a9, 	0,		0];
											
// master grip angle fitting coefficients(wrt normalized hall sensor value)
g_masterGripAngleFitCoeff2 : ARRAY[1..4] OF LREAL :=
	[2383.519457, -348.6613075, -3.070925, 0.5172933123];
g_masterGripAngleFitCoeff : ARRAY[1..6] OF LREAL :=
	[4.013978, -10.454747, 9.464741, -3.7829344, 0.447868, 0.339937];
g_maxGripAngle : LREAL := 30.0 * g_deg2Rad;
g_minGripAngle :LREAL  := 0.0;

END_VAR

// ---- GVLs/GVL_SafetyParameters.TcGVL
{attribute 'global_init_slot' := '49991'}
//TODO: safety check parameters need to be reviewd
VAR_GLOBAL CONSTANT
	
	// safety error counts threshold to trigger fault
	g_faultTriggerCounts :INT :=2;
	
	// arm joint safety error
	g_armMaxJntEncErr :vec7d:=[7(40*g_deg2Rad)];
	g_armMaxJntFollowErr :vec7d:=[7(20*g_deg2Rad)];
	
	// joint limit buffer(outside of joint limit)
	g_armJntPosLimitBuffer :vec7d:=[3(10.0*g_deg2Rad), 4(45.0*g_deg2Rad)];

	//max joint encoder current  saltation
	g_maxJntCurSalta : vec7di:=[7(60000)];
	
	// self check timeout time limit
	g_selfCheckTimeLimit : LREAL:= 15.0;
	
	//arm joint link encoder maximum and minimum values
	g_maxLinkEnc : DINT:=16777215;
	g_minLinkEnc : DINT:=0;
	
	//drive error word
	g_driveErrWord : UDINT:=32;
	
	// master arm cartesion control safety error 
	g_maxCartPosErr :LREAL := 0.005;
	g_maxCartOriErr :LREAL := 5.0*g_deg2Rad;
	

	// master joint safety error
	g_maxJntCtrlErr :LREAL := 15.0*g_deg2Rad;
	g_maxJntEncErr :LREAL := 30.0*g_deg2Rad;
	
	g_minJntPos: ARRAY[1..2,1..7] OF LREAL:=[-60*g_deg2Rad,	-45*g_deg2Rad-pi/2,		-45*g_deg2Rad, 	0, 	-135*g_deg2Rad+pi,		-60*g_deg2Rad-pi/2,		-g_largeNum,
											 -60*g_deg2Rad,	-45*g_deg2Rad-pi/2,		-45*g_deg2Rad,	0,		-135*g_deg2Rad+pi,		-60*g_deg2Rad+pi/2-pi,	-g_largeNum];
	g_maxJntPos: ARRAY[1..2,1..7] OF LREAL:=[60*g_deg2Rad,	60*g_deg2Rad-pi/2,		60*g_deg2Rad,		2*pi,			135*g_deg2Rad+pi,		60*g_deg2Rad-pi/2+pi,		g_largeNum,
								             60*g_deg2Rad,	60*g_deg2Rad-pi/2,		60*g_deg2Rad,		2*pi,			135*g_deg2Rad+pi,		60*g_deg2Rad+pi/2,		g_largeNum];

	
	// cart joint safety error
	g_cartMaxJntCtrlErr :Vec4d := [0.005, 5*g_deg2Rad,0.005, 0.005];
	g_cartMaxJntEncErr :Vec4d :=  [0.005, 5*g_deg2Rad,0.005, 0.005];

	// cart joint limit buffer(outside of joint limit)
	g_cartJntPosLimitBuffer :Vec4d :=[0.05, 10*g_deg2Rad,0.05, 0.05];
	
	// cart joint velocity limit
	g_cartMaxJntVel :Vec4d :=[0.03, 4*g_deg2Rad,0.02,0.015];
	
	// cart joint limit
	g_cartMinJntLimit : Vec4d :=[0-0.1, -(38+5)*g_deg2Rad, 0-0.1, 0-0.1];
	g_cartMaxJntLimit : Vec4d :=[0.4+0.1, (12+5)*g_deg2Rad, 0.3+0.1, 0.2+0.1];
	
	
	//cart joint follow error
	g_cartMaxJntFollowErr : Vec4d :=[0.01, 5*g_deg2rad, 0.01, 0.01];
	
	//cart joint current limit
	g_cartMaxJntCurrent : Vec4d :=[3800*2,3800*2,3800*2,3800*2];
	
	//cart joint encoder detetion value
	g_cartMaxLinkEnc : ARRAY [1..4] OF DINT := [67108863,16777215,67108863,67108863];
	g_cartMinLinkEnc : ARRAY [1..4] OF DINT := [4(0)];
END_VAR

VAR_GLOBAL
	//motor current limit
	g_motorCurrentLimit : Vec7d ;	

	g_arrayErrCodeArm:ARRAY [1..g_maxNum] OF ARRAY [0..100] OF UDINT;	
	
	g_ArrayErrCodeTypeTest:ARRAY [1..3] OF ARRAY [0..100] OF UDINT;
END_VAR

VAR_GLOBAL CONSTANT
	g_maxNum:INT:=3;
	g_maxArmNum:INT:=2;
	g_maxArmJoint:INT:=7; g_maxCartJoint:INT:=4;
	g_cartNum:UDINT:=3;
	MAX_CSV_ROWS 			: UDINT := 10000;(*最大行数(任务周期为20ms)即10分钟的buffer*)
	MAX_CSV_COLUMNS 		: UDINT := 130;(*最大列数*)
	MAX_CSV_FIELD_LENGTH	: UDINT := 35;(*每个字段的字符长度*)
	MAX_CSV_RING_BUFFER		: UDINT := 3;
	g_ArmNetID: ARRAY[1..g_maxArmNum] OF T_AmsNetId:=['169.254.79.95.2.1','169.254.219.236.5.1'];
	g_JointNetPort:ARRAY[1..g_maxArmNum,1..g_maxArmJoint] OF UINT :=[
											1001,    1001,	1002,	1003,	1004,	1005,	1006,
											1011,    1011,	1012,	1013,	1014,	1015,	1016	];
	g_cartNetID : T_AmsNetId := '169.254.219.236.5.1';
	g_cartJointNetPort:ARRAY[1..g_maxCartJoint] OF UINT :=[1007,    1008,	1009,	1010];
	
END_VAR

// ---- FBs_Auxiliary/FB_GripAngleCalc.TcPOU
FUNCTION_BLOCK FB_GripAngleCalc
VAR_INPUT
END_VAR
VAR_OUTPUT
END_VAR
VAR
	// limit value
	m_minHallSensorValue :LREAL;
	m_maxHallSensorValue:LREAL;
	m_hallSensorRange:LREAL;
	
	// grip angle from hall sensor IO
	m_gripHallSenorValue :LREAL;
	m_normHallSensorValue: LREAL;
	m_gripAngle :LREAL;
	m_gripAngLpf : FB_LowPassFilter;
END_VAR

METHOD init : BOOL
VAR_INPUT
	i_armIdx:INT;
END_VAR
// init limit value
m_minHallSensorValue:=(GVL_ArmJointCaliData.g_minHallSensorValue[i_armIdx]/65536) AND 16#0000FFFF; 
m_maxHallSensorValue:=(GVL_ArmJointCaliData.g_maxHallSensorValue[i_armIdx]/65536) AND 16#0000FFFF; 
m_hallSensorRange := m_maxHallSensorValue-m_minHallSensorValue;

// init filter
m_gripAngLpf.init(1, g_gripAngLpfCutoffFreq, g_armCtrlFreq);
END_METHOD

METHOD run : LREAL
VAR_INPUT
	IOValue : UDINT;
END_VAR
// sensor io parse
m_gripHallSenorValue:=(IOValue/65536) AND 16#0000FFFF; //high 16 bits

// normalize hall sensor value
m_normHallSensorValue:=LIMIT(0, (m_gripHallSenorValue-m_minHallSensorValue)/m_hallSensorRange, 1);

m_gripAngle := g_masterGripAngleFitCoeff[1] * EXPT(m_normHallSensorValue,5)
		+ g_masterGripAngleFitCoeff[2] * EXPT(m_normHallSensorValue,4)
		+ g_masterGripAngleFitCoeff[3] * EXPT(m_normHallSensorValue,3)
		+ g_masterGripAngleFitCoeff[4] * EXPT(m_normHallSensorValue,2)
		+ g_masterGripAngleFitCoeff[5] * EXPT(m_normHallSensorValue,1)
		+ g_masterGripAngleFitCoeff[6];

// filt and cap the result
m_gripAngle := m_gripAngLpf.run(m_gripAngle);
m_gripAngle := LIMIT(g_minGripAngle, m_gripAngle, g_maxGripAngle);

run:=m_gripAngle;
END_METHOD

END_FUNCTION_BLOCK

// ---- FBs_Robots/FB_CartJoint.TcPOU
FUNCTION_BLOCK FB_CartJoint EXTENDS FB_JointBase
VAR_INPUT
END_VAR
VAR_OUTPUT
END_VAR
VAR
END_VAR

METHOD PUBLIC init : BOOL
VAR_INPUT
	i_jntIdx :INT;
	i_controlCycleTime :LREAL;
END_VAR
m_cycleTime := i_controlCycleTime;

// hardware parameters
m_motorEncoderRes :=GVL_CartJointParameters.g_incEncoderRes[i_jntIdx];
m_linkEncoderRes :=GVL_CartJointParameters.g_absEncoderRes[i_jntIdx];
m_motorReduction :=GVL_CartJointParameters.g_motorReduction[i_jntIdx];
m_linkEncoderReduction :=GVL_CartJointParameters.g_absEncoderReduction[i_jntIdx];
m_trqConst :=GVL_CartJointParameters.g_motorTrqConst[i_jntIdx];
m_maxCurrent :=GVL_CartJointParameters.g_motorMaxCurrent[i_jntIdx];
m_motorDir :=GVL_CartJointParameters.g_motorDir[i_jntIdx];								
m_linkEncoderDir :=GVL_CartJointParameters.g_asbEncoderDir[i_jntIdx];
m_minJntPos	:=GVL_CartJointParameters.g_minJntPos[i_jntIdx];
m_maxJntPos	:=GVL_CartJointParameters.g_maxJntPos[i_jntIdx];

//link encoder calibartion data
m_minLinkEncoder :=GVL_CartJointCaliData.g_minLinkEncoder[i_jntIdx] - m_linkEncoderDir*GVL_CartJointCaliData.g_linkEncLimitBuffer[i_jntIdx]; // expand limit
m_maxLinkEncoder :=GVL_CartJointCaliData.g_maxLinkEncoder[ i_jntIdx] + m_linkEncoderDir*GVL_CartJointCaliData.g_linkEncLimitBuffer[i_jntIdx]; // expand limit
m_caliLinkEncoder :=GVL_CartJointCaliData.g_caliLinkEncoder[i_jntIdx];
m_linkEncCaliJntPos :=GVL_CartJointCaliData.g_linkEncCaliJntPos[i_jntIdx];
m_linkEncZeroCross :=GVL_CartJointCaliData.g_linkEncZeroCross[i_jntIdx];
m_multiCycles :=GVL_CartJointCaliData.g_multipleCyclesJoint[i_jntIdx];

// convert cali link encoder if joint cross zero
IF 1=m_linkEncZeroCross THEN
	IF 1=m_linkEncoderDir AND m_caliLinkEncoder < m_minLinkEncoder THEN
		m_caliLinkEncoder := GVL_CartJointCaliData.g_caliLinkEncoder[i_jntIdx] + m_linkEncoderRes;
	ELSIF -1=m_linkEncoderDir AND m_caliLinkEncoder < m_maxLinkEncoder THEN
		m_caliLinkEncoder := GVL_CartJointCaliData.g_caliLinkEncoder[i_jntIdx] + m_linkEncoderRes;
	END_IF
END_IF

// macro data
m_trq2CurrentRatio:=m_motorDir * 1000.0/(m_trqConst*m_motorReduction);
m_current2TrqRatio:=m_motorDir * (m_trqConst*m_motorReduction)/1000.0;
m_linkEnc2PosRatio := 2*PI*m_linkEncoderDir/(m_linkEncoderReduction*m_linkEncoderRes);
m_motorEnc2PosRatio := 2*PI * m_motorDir/(m_motorReduction * m_motorEncoderRes);

// motor data init
m_curJntVel:=0;
m_curJntTrq :=0;
m_rawCurrent :=0;
m_filtCurrent :=0;
m_cmdJntVel :=0.0;
m_cmdJntTrq :=0.0;
m_cmdCurrent := 0.0;

// filter init
m_jntVelLpf.init(1, g_curJntVelLpfCutoffFreq, g_cartCtrlFreq);
m_linkVelLpf.init(1, g_curJntVelLpfCutoffFreq, g_cartCtrlFreq);
m_cmdTrqLpf.init(1, g_cmdJntTrqLpfCutoffFreq, g_cartCtrlFreq);
m_curTrqLpf.init(1, g_curJntTrqLpfCutoffFreq, g_cartCtrlFreq);

// driver init value
m_motorOutputs.m_controlWord:=DriverCtrlWord_INIT;
m_motorOutputs.m_opMode:=INT_TO_SINT(DriverOPMode_Pos);
m_motorOutputs.m_cmdCurrent:=0;
m_motorOutputs.m_cmdMotorEncoder:=m_motorInputs.m_motorEncoder;
END_METHOD

END_FUNCTION_BLOCK

// ---- FBs_Robots/FB_JointBase.TcPOU
FUNCTION_BLOCK FB_JointBase
VAR
	// motor IO
	m_motorInputs AT%I*	:ST_MotorInputs;
	m_motorOutputs AT%Q* :ST_MotorOutputs;
		
	// cycle time
	m_cycleTime :LREAL;
	
	// calibrated link encoder data
	m_minLinkEncoder :DINT;
	m_maxLinkEncoder :DINT;
	m_caliLinkEncoder :DINT;
	m_linkEncCaliJntPos :LREAL;
	m_linkEncZeroCross :INT;
	m_initMotorEnc : DINT;
	m_multiCycles :INT;
	
	// joint position from link encoder after power on
	m_initLinkPos :LREAL;
	
	// data for link encoder multiple cycles
	m_lastLinkEncoder :DINT;
	m_linkEncCycles:INT;
	
	// device paramters
	m_motorEncoderRes :DINT;
	m_linkEncoderRes :DINT;
	m_motorReduction :LREAL;
	m_linkEncoderReduction :LREAL;
	m_trqConst :LREAL;
	m_maxCurrent :LREAL;
	m_motorDir :INT;								
	m_linkEncoderDir :INT;
	m_minJntPos: LREAL;
	m_maxJntPos: LREAL;
	
	// macro defined data for quick calculation
	m_trq2CurrentRatio:LREAL;
	m_current2TrqRatio:LREAL;
	m_linkEnc2PosRatio :LREAL;
	m_motorEnc2PosRatio :LREAL;
	
	// joint data
	m_curMotorPos :LREAL;
	m_curLinkPos :LREAL;
	m_curJntPos	:LREAL;
	m_curJntVel :LREAL;
	m_curLinkVel :LREAL;
	m_curJntTrq :	LREAL;
	m_rawCurrent : LREAL;
	m_filtCurrent : LREAL;
	m_cmdJntPos :LREAL;
	m_cmdJntVel :LREAL;
	m_cmdJntTrq :LREAL;
	m_cmdCurrent : LREAL;
	m_lastJntPos :LREAL;
	m_lastLinkPos: LREAL;
	
	// velocity filter
	m_jntVelLpf :FB_LowPassFilter;
	m_linkVelLpf :FB_LowPassFilter;
	
	// current and command torque filter
	m_curTrqLpf : FB_LowPassFilter;
	m_cmdTrqLpf :FB_LowPassFilter;
	
		newLinkEnc :DINT;
END_VAR

PROPERTY cmdCurrent : LREAL
GET
cmdCurrent:=m_cmdCurrent;
END_GET
END_PROPERTY

METHOD PUBLIC disable : BOOL
VAR_INPUT
END_VAR
m_motorOutputs.m_controlWord:=DriverCtrlWord_INIT;
disable:=true;
END_METHOD

METHOD PUBLIC enable : BOOL
VAR_INPUT
END_VAR
IF DriverStatusWord_INIT = m_motorInputs.m_statusWord THEN
	m_motorOutputs.m_controlWord:=DriverCtrlWord_PREOP;
	enable := FALSE;
ELSIF DriverStatusWord_PREOP = m_motorInputs.m_statusWord THEN
	m_motorOutputs.m_controlWord:=DriverCtrlWord_OP;
	enable :=  FALSE;
ELSIF DriverStatusWord_OP = m_motorInputs.m_statusWord THEN
	enable :=  TRUE;
//ELSE
//	m_motorOutputs.m_controlWord:=DriverCtrlWord_INIT;
//	enable :=  FALSE;
END_IF
END_METHOD

PROPERTY filtCurrent : LREAL
GET
filtCurrent:=m_filtCurrent;
END_GET
END_PROPERTY

METHOD PUBLIC initJntPos : BOOL
VAR_INPUT
END_VAR
m_lastLinkEncoder :=m_motorInputs.m_linkEncoder;
m_linkEncCycles:=0;
m_curLinkPos :=linkEnc2Pos();
m_initLinkPos:=m_curLinkPos;
m_initMotorEnc :=m_motorInputs.m_motorEncoder;
m_curMotorPos:=motorEnc2Pos();
m_curJntPos := m_curMotorPos;
m_cmdJntPos :=m_curJntPos;	
m_lastJntPos :=m_curJntPos;
m_lastLinkPos := m_curLinkPos;

// filter init
m_jntVelLpf.init(1, g_curJntVelLpfCutoffFreq, g_armCtrlFreq);
m_linkVelLpf.init(1, g_curJntVelLpfCutoffFreq, g_armCtrlFreq);
END_METHOD

// reset the initial joint position with input value
METHOD PUBLIC initJntPosReset : BOOL
VAR_INPUT
	i_initLinkPos:LREAL;
END_VAR
m_initLinkPos:=i_initLinkPos;
m_initMotorEnc :=m_motorInputs.m_motorEncoder;
m_curMotorPos:=motorEnc2Pos();
m_curJntPos := m_curMotorPos;
m_cmdJntPos :=m_curJntPos;	
m_lastJntPos :=m_curJntPos;
m_lastLinkPos := m_curLinkPos;

// filter init
m_jntVelLpf.init(1, g_curJntVelLpfCutoffFreq, g_armCtrlFreq);
m_linkVelLpf.init(1, g_curJntVelLpfCutoffFreq, g_armCtrlFreq);
END_METHOD

PROPERTY initLinkPos : lreal
GET
initLinkPos:=m_initLinkPos;
END_GET
SET
//m_initLinkPos:=initLinkPos;
END_SET
END_PROPERTY

METHOD PUBLIC isEnabled : BOOL
VAR_INPUT
END_VAR
isEnabled :=(DriverStatusWord_OP = m_motorInputs.m_statusWord);
END_METHOD

PROPERTY jntPos : LREAL
GET
jntPos := m_curJntPos;
END_GET
END_PROPERTY

PROPERTY jntTrq : LREAL
GET
jntTrq:=m_curJntTrq;
END_GET
END_PROPERTY

PROPERTY jntVel : LREAL
GET
jntVel := m_curJntVel;
END_GET
END_PROPERTY

METHOD PROTECTED linkEnc2Pos : LREAL
VAR_INPUT
END_VAR
VAR
	incLinkPos :LREAL;

END_VAR
// cycle check
IF 1=m_multiCycles THEN
	IF (m_motorInputs.m_linkEncoder - m_lastLinkEncoder)*m_linkEncoderDir < -m_linkEncoderRes/2 THEN
		m_linkEncCycles :=m_linkEncCycles+1;
	ELSIF (m_motorInputs.m_linkEncoder - m_lastLinkEncoder)*m_linkEncoderDir > m_linkEncoderRes/2 THEN
		m_linkEncCycles :=m_linkEncCycles-1;
	END_IF
END_IF
m_lastLinkEncoder:=m_motorInputs.m_linkEncoder;

// convert link encoder if joint cross zero
newLinkEnc := m_motorInputs.m_linkEncoder;
IF 1=m_linkEncZeroCross AND 0 = m_multiCycles THEN
	IF 1=m_linkEncoderDir AND m_motorInputs.m_linkEncoder < m_minLinkEncoder THEN
		newLinkEnc := m_motorInputs.m_linkEncoder + m_linkEncoderRes;
	ELSIF -1=m_linkEncoderDir AND m_motorInputs.m_linkEncoder < m_maxLinkEncoder THEN
		newLinkEnc := m_motorInputs.m_linkEncoder + m_linkEncoderRes;
	END_IF
END_IF

// motion from calibrated points
incLinkPos := (newLinkEnc-m_caliLinkEncoder)*m_linkEnc2PosRatio;

// absolute joint position
linkEnc2Pos := incLinkPos + m_linkEncCaliJntPos + 2*PI* m_linkEncCycles;
END_METHOD

PROPERTY PUBLIC linkPos : LREAL
GET
linkPos:=m_curLinkPos;
END_GET
END_PROPERTY

METHOD PROTECTED motorEnc2Pos : LREAL
VAR_INPUT
END_VAR
motorEnc2Pos:= (m_motorInputs.m_motorEncoder-m_initMotorEnc)* m_motorEnc2PosRatio +m_initLinkPos;
END_METHOD

PROPERTY PUBLIC motorPos : LREAL
GET
motorPos := m_curMotorPos;
END_GET
END_PROPERTY

METHOD PROTECTED motorPos2Enc : DINT
VAR_INPUT
	i_jntPos :LREAL;
END_VAR

VAR
END_VAR
motorPos2Enc := LREAL_TO_DINT((i_jntPos-m_initLinkPos)/m_motorEnc2PosRatio + m_initMotorEnc);
END_METHOD

PROPERTY rawCurrent : LREAL
GET
rawCurrent := m_rawCurrent;
END_GET
END_PROPERTY

METHOD PUBLIC updateCmds : BOOL
VAR_INPUT
	i_opMode : E_DriverOPMode;
	i_cmdPos :LREAL;
	i_cmdTrq :LREAL;
END_VAR
VAR
	filtCmdTrq :LREAL;
END_VAR
m_motorOutputs.m_opMode:=INT_TO_SINT( i_opMode);
// pos mode
IF i_opMode = DriverOPMode_Pos THEN
	m_motorOutputs.m_cmdCurrent:=0;
	m_cmdTrqLpf.reset();
//	i_cmdPos:=LIMIT(m_minJntPos, i_cmdPos, m_maxJntPos);
	m_motorOutputs.m_cmdMotorEncoder :=motorPos2Enc(i_cmdPos);
ELSIF i_opMode = DriverOPMode_Trq THEN
	filtCmdTrq:=m_cmdTrqLpf.run(i_cmdTrq);
	m_motorOutputs.m_cmdCurrent:=LREAL_TO_DINT(LIMIT(-m_maxCurrent, filtCmdTrq*m_trq2CurrentRatio,m_maxCurrent));
	m_motorOutputs.m_cmdMotorEncoder :=m_motorInputs.m_motorEncoder; 
END_IF
m_cmdCurrent:=m_motorOutputs.m_cmdCurrent;
END_METHOD

METHOD PUBLIC updateStatus : BOOL
VAR_INPUT
END_VAR
// compute joint position
m_curLinkPos:= linkEnc2Pos();
m_curMotorPos:=motorEnc2Pos();
m_curJntPos := m_curMotorPos;

// compute joint velocity
m_curJntVel:= (m_curJntPos-m_lastJntPos)/m_cycleTime;
m_curJntVel := m_jntVelLpf.run(m_curJntVel);
m_lastJntPos :=m_curJntPos;

// compute link velocity
m_curLinkVel := (m_curLinkPos-m_lastLinkPos)/m_cycleTime;
m_curLinkVel := m_linkVelLpf.run(m_curLinkVel);
m_lastLinkPos := m_curLinkPos;

// current and torque
m_rawCurrent := m_motorInputs.m_current;
m_filtCurrent := m_curTrqLpf.run(m_rawCurrent);
m_curJntTrq := m_filtCurrent * m_current2TrqRatio;
END_METHOD

END_FUNCTION_BLOCK

// ---- FBs_Robots/FB_MasterCart.TcPOU
FUNCTION_BLOCK FB_MasterCart
VAR
	//  IO and check
	m_endoScopePedalIO AT%I* :BOOL;
	m_endoScopeIOCheck :FB_IOCheck;
	
	m_clutchPedalIO AT%I* :BOOL;
	m_clutchIOCheck :FB_IOCheck;
	
	m_surgonHeadInIO AT%I* :BOOL;
	m_headInCheck:FB_IOCheck;
	
	m_armSwitchIO AT%I* :BOOL;
	m_armSwitchCheck:FB_IOToggleCheck;
	
	m_electricCutLeft AT %I* :BOOL;
	m_electricCutLeftAllow AT %I* :BOOL;
	
	m_electricCutRight AT %I* :BOOL;
	m_electricCutRightAllow AT %I* :BOOL;
	
	m_electricCoagulLeft AT %I* :BOOL;
	m_electricCoagulLeftAllow AT %I* :BOOL;
	
	m_electricCoagulRight AT %I* :BOOL;
	m_electricCoagulRightAllow AT %I* :BOOL;
	
	m_elecKnifeCtrlWord AT %Q* :DINT;
	
	// cart status
	m_cartStatus  : ST_CartStatus;
	
	// cart joints
	// [monitor lift, monitor rotate, armset, pedal]
	m_cartJoints:ARRAY[1..4] OF FB_CartJoint;
	
	// cart joint motion control IO
	//[monitor_up, monitor_down, monitor_cwRotate, monitor_ccwRotate, armset_up, armset_down, pedal_in, pedal_out]
	m_cartJointCtrlIO AT%I* :ARRAY[1..8] OF BOOL ;
	m_cartJointCtrlIOCheck :ARRAY[1..8] OF FB_IOCheck;
	
	//electrotome control io
	m_electricCutLeftOn :BOOL;
	m_electricCutRightOn :BOOL;
	m_electricCoagulLeftOn : BOOL;
	m_electricCoagulRightOn : BOOL;
	//Triggering several energies at once
	m_eleCtrlState : UINT;
	//The type of instrument energy of the master hand corresponding to the slave hand
	m_energyType :ARRAY[1..g_mArmNum] OF UINT :=[2(0)];
	
	// cart joint control data
	m_jntEnableCounts:Vec4i ;
	m_jntDisableCounts:Vec4i ;
	m_jntEnableCountsThres:INT:=500;
	m_jntCmdMotionDir :Vec4i;
	m_cmdJntTrq :Vec4d;
	m_cmdJntPos :Vec4d;
	m_cmdJntVel :Vec4d;
	m_jntEnableFlag :Vec4b;
	
	//cart ergonomic adjust data
	m_UIData : ST_CartUIData;
	m_carInMotion : INT; // 0:  no mition, 1: mamual adjust, 2: ergonomic adjust
	m_jntSoftwareLimit :ARRAY [1..4] OF LREAL := [0.01, 1*g_deg2Rad, 0.015, 0.005];
	m_cmdArrival : Vec4b;
	
	// cart joint status data
	m_curMotorPos :Vec4d;
	m_curLinkPos :Vec4d;
	m_curJntPos :Vec4d;
	m_curJntVel :Vec4d;
	m_curJntTrq :Vec4d;
	m_rawJntCurrent :Vec4d;
	m_filtJntCurrent :Vec4d;
	m_cmdJntCurrent : Vec4d;

END_VAR

METHOD eleKnifeCtrl : DINT
VAR_IN_OUT CONSTANT
	m_armState:ARRAY[1..g_mArmNum] OF E_masterArmState ;
	m_teleSlaveArmIdx :ARRAY[1..g_mArmNum] OF E_MatchedSlaveArmIdx;
	m_instruStauts: ARRAY[1..g_sArmNum] OF ST_InstruStatus;
END_VAR
//Foot trigger check
m_electricCutLeftOn := m_electricCutLeft AND m_electricCutLeftAllow AND m_armState[1] = MasterArmState_MasterSlave ;
m_electricCutRightOn := m_electricCutRight AND m_electricCutRightAllow AND m_armState[2] = MasterArmState_MasterSlave ;
m_electricCoagulLeftOn := m_electricCoagulLeft AND m_electricCoagulLeftAllow AND m_armState[1] = MasterArmState_MasterSlave ;
m_electricCoagulRightOn := m_electricCoagulRight AND m_electricCoagulRightAllow AND m_armState[2] = MasterArmState_MasterSlave ;

//You cannot excite two energies at the same time
m_eleCtrlState := BOOL_TO_UINT(m_electricCutLeftOn) + BOOL_TO_UINT(m_electricCutRightOn)
										 + BOOL_TO_UINT(m_electricCoagulLeftOn) + BOOL_TO_UINT(m_electricCoagulRightOn);

IF m_teleSlaveArmIdx[1] > 0 THEN
	m_energyType[1] := m_instruStauts[m_teleSlaveArmIdx[1]].m_energyType;
	m_energyType[2] := m_instruStauts[m_teleSlaveArmIdx[2]].m_energyType;
END_IF

IF m_eleCtrlState = 1 THEN
	IF (m_electricCutLeftOn AND  m_energyType[1] = InstruType_isMonopole) OR (m_electricCutRightOn AND  m_energyType[2] = InstruType_isMonopole) THEN
		eleKnifeCtrl := EnergyCtrlWord_isMonopoleCut;
	ELSIF (m_electricCoagulLeftOn AND m_energyType[1] = InstruType_isMonopole) OR (m_electricCoagulRightOn AND  m_energyType[2] = InstruType_isMonopole) THEN
		eleKnifeCtrl := EnergyCtrlWord_isMonopoleCoagul;
	ELSIF (m_electricCoagulLeftOn AND m_energyType[1] = InstruType_isBipolar) OR (m_electricCoagulRightOn AND  m_energyType[2] = InstruType_isBipolar) THEN
		eleKnifeCtrl := EnergyCtrlWord_isBipolarCoagul;
	ELSIF (m_electricCutLeftOn AND m_energyType[1] = InstruType_isUltraKnife) OR (m_electricCutRightOn AND  m_energyType[2] = InstruType_isUltraKnife) THEN
		eleKnifeCtrl := EnergyCtrlWord_isUltraMin;
	ELSIF (m_electricCoagulLeftOn AND m_energyType[1] = InstruType_isUltraKnife) OR (m_electricCoagulRightOn AND  m_energyType[2] = InstruType_isUltraKnife) THEN
		eleKnifeCtrl := EnergyCtrlWord_isUltraMax;
		
	ELSE
		eleKnifeCtrl := EnergyCtrlWord_NoOutput;
	END_IF
ELSE
	eleKnifeCtrl := EnergyCtrlWord_NoOutput;
END_IF
END_METHOD

METHOD ergonomicAdjust : INT
VAR_INPUT
END_VAR
VAR
	i : INT;
	err:Vec4d;
END_VAR
vecSub(m_UIData.m_cmdJntPos,m_curJntPos, err);
ergonomicAdjust := 2;
//only update command after joints is truly enabled
FOR i := 1 TO 4 DO
	IF m_jntEnableFlag[i] AND m_cartJoints[i].isEnabled() AND m_jntEnableCounts[i]>= m_jntEnableCountsThres THEN
		m_cmdJntVel[i]:=sign(m_UIData.m_cmdJntPos[i]-m_cartJoints[i].jntPos)*(GVL_CartJointParameters.g_jntCtrlMotionVel[i]);
		IF ABS(err[i]) < m_jntSoftwareLimit[i]/3 THEN
			m_cmdJntVel[i]:=0;
		END_IF
		m_cmdJntPos[i] := LIMIT(GVL_CartJointParameters.g_minJntPos[i] + m_jntSoftwareLimit[i],  m_cmdJntPos[i] + m_cmdJntVel[i]*g_cartCtrlCycleTime, GVL_CartJointParameters.g_maxJntPos[i] - m_jntSoftwareLimit[i]);
	
	ELSE
		m_cmdJntVel[i]:=0;
		m_cmdJntPos[i] := m_cartJoints[i].jntPos;
	END_IF	
END_FOR
END_METHOD

METHOD PUBLIC getStatus : BOOL
VAR_IN_OUT
	// cart status data
	r_cartStatus :ST_CartStatus;
	
	// cart joint data
	r_cartJointData :ST_CartJointData;
	
END_VAR
r_cartStatus := m_cartStatus;


// current joint data
r_cartJointData.m_curMotorPos:=m_curMotorPos;
r_cartJointData.m_curLinkPos:=m_curLinkPos;
r_cartJointData.m_curJntPos:=m_curJntPos;
r_cartJointData.m_curJntVel:=m_curJntVel;
r_cartJointData.m_curJntTrq:=m_curJntVel;
r_cartJointData.m_rawJntCurrent:=m_rawJntCurrent;
r_cartJointData.m_filtJntCurrent:=m_filtJntCurrent;

// command joint data
r_cartJointData.m_cmdJntPos:=m_cmdJntPos;
r_cartJointData.m_cmdJntVel:=m_cmdJntVel;
r_cartJointData.m_cmdJntTrq:=m_cmdJntTrq;
r_cartJointData.m_cmdJntCurrent:=m_cmdJntCurrent;
END_METHOD

METHOD PUBLIC init : BOOL
VAR_INPUT
END_VAR
VAR
	i:INT;
	initLinkPos :LREAl;
END_VAR
// joint init
FOR i:=1 TO 4 DO
	m_cartJoints[i].init(i,g_cartCtrlCycleTime);
	m_cartJoints[i].initJntPos();
END_FOR

// motor and link encoder of  monitor rotation are on different  joints
// transfer monitor angle from link side to motor side
initLinkPos:= monitorAngLink2Motor(m_cartJoints[2].initLinkPos);
m_cartJoints[2].initJntPosReset(initLinkPos);

// init commands
FOR i:=1 TO 4 DO
	m_jntEnableCounts[i]:=0;
	m_jntDisableCounts[i]:=0;
	m_jntEnableFlag[i]:=FALSE;
	m_jntCmdMotionDir[i]:=0;
	m_cmdJntTrq[i]:=0;
	m_cmdJntVel[i]:=0;
	m_cmdJntPos[i]:=m_cartJoints[i].jntPos;
END_FOR

m_cartStatus.m_initFlag :=true;
END_METHOD

METHOD manualAdjust : INT
VAR_INPUT
END_VAR
VAR
	i : INT;
END_VAR
// update joint command positon
manualAdjust := 1;
//only update command after joints is truly enabled
FOR i := 1 TO 4 DO
	IF  m_jntEnableFlag[i] AND m_cartJoints[i].isEnabled() AND m_jntEnableCounts[i]>= m_jntEnableCountsThres THEN
		//  update command joint velocity
		m_cmdJntVel[i]:=m_jntCmdMotionDir[i]*GVL_CartJointParameters.g_jntCtrlMotionVel[i];
		
		// limit handle
		IF (m_cmdJntPos[i]> GVL_CartJointParameters.g_maxJntPos[i] - m_jntSoftwareLimit[i] AND m_cmdJntVel[i] >0 ) OR 
				(m_cmdJntPos[i]< GVL_CartJointParameters.g_minJntPos[i] + m_jntSoftwareLimit[i] AND m_cmdJntVel[i] <0 )  THEN
				m_cmdJntVel[i] := 0.0;
		END_IF
		m_cmdJntPos[i]:= m_cmdJntPos[i]+ m_cmdJntVel[i]*g_cartCtrlCycleTime;
	ELSE
		m_cmdJntVel[i]:=0;
		m_cmdJntPos[i] := m_cartJoints[i].jntPos;
	END_IF
END_FOR
END_METHOD

// TODO
METHOD PROTECTED monitorAngLink2ImagiAxis : LREAL
VAR_INPUT
	i_linkPos:LREAL;
END_VAR
VAR
	A,B,C,D,E,F,G,H,I,X0,X1,X2,X3,X4,X5,X6,X7,X8,X9,X10,X11,X12,Z0:LREAL;	
END_VAR

X0:=i_linkPos;  //监视器旋转

A:=222; B:=191.5; C:=232.7073; D:=135.5031; E:=186; F:=164; G:=178; H:=45; I:=160;
X4:=ATAN(H/I); X5:=ATAN(F/G);
X8:=SQRT(F*F+G*G);
X12:=sqrt(H*H+I*I);
X9:=sqrt(E*E+X12*X12-2*E*X12*cos(X0));
X6:=acos((B*B+X8*X8-X9*X9)/(2*B*X8));
X10:=acos((B*B+X9*X9-X8*X8)/(2*B*X9));
X11:=acos((X9*X9+X12*X12-E*E)/(2*X9*X12));
X7:=X10+X11;
X2:=X5-X6;
X3:=pi-X7+X2;
X1:=X3-X4;

monitorAngLink2ImagiAxis:=X1;
END_METHOD

// TODO
METHOD PROTECTED monitorAngLink2Motor : LREAL
VAR_INPUT
	i_linkPos:LREAL;
END_VAR
VAR
	A,B,C,D,E,F,G,H,I,X0,X1,X2,X3,X4,X5,X6,X7,X8,X9,X10,X11,X12,Z0:LREAL;	
END_VAR

X0:=i_linkPos;  //监视器旋转

A:=222; B:=191.5; C:=232.7073; D:=135.5031; E:=186; F:=164; G:=178; H:=45; I:=160;
X4:=ATAN(H/I); X5:=ATAN(F/G);
X8:=SQRT(F*F+G*G);
X12:=sqrt(H*H+I*I);
X9:=sqrt(E*E+X12*X12-2*E*X12*cos(X0));
X6:=acos((B*B+X8*X8-X9*X9)/(2*B*X8));
X10:=acos((B*B+X9*X9-X8*X8)/(2*B*X9));
X11:=acos((X9*X9+X12*X12-E*E)/(2*X9*X12));
X7:=X10+X11;
X2:=X5-X6;
X3:=pi-X7+X2;
X1:=X3-X4;

monitorAngLink2Motor:=X2;
END_METHOD

//TODO
METHOD PROTECTED monitorAngMotor2Link : LREAL
VAR_INPUT
	i_motorPos:LREAL;
END_VAR
VAR
	A,B,C,D,E,F,G,H,I,X0,X1,X2,X3,X4,X5,X6,X7,X8,X9,X10,X11,X12,Z0:LREAL;	
END_VAR
X2:=i_motorPos;

A:=222; B:=191.5; C:=232.7073; D:=135.5031; E:=186; F:=164; G:=178; H:=45; I:=160;
X5:=atan(F/G);
X6:=X5-X2;
X8:=sqrt(F*F+G*G);
X9:=sqrt(B*B+X8*X8-2*B*X8*cos(X6));
X12:=SQRT(H*H+I*I);
X0:=ACOS((E*E+X12*X12-X9*X9)/(2*E*X12));

monitorAngMotor2Link:=X0;
END_METHOD

METHOD reachUITargetCheck : bool
VAR
	i :INT;
	err:Vec4d;
END_VAR
vecSub(m_UIData.m_cmdJntPos,m_curJntPos, err);

// joint error check
FOR i:=1 TO 4 DO 
	m_cmdArrival[i] :=  ABS(err[i]) < m_jntSoftwareLimit[i]/2;
END_FOR
END_METHOD

METHOD PUBLIC run : BOOL
VAR_IN_OUT CONSTANT
	i_cartUIData : ST_CartUIData;
END_VAR
VAR
	i:INT;
END_VAR
// update IO signals
updateIO(i_cartUIData);

// update cart status
updateStatus();

// update controller and command
updateCmds();

// send command to joint driver
FOR i:=1 TO 4 DO
	// joint enable
	IF m_jntEnableFlag[i] AND NOT(SafetyCheck.m_safetyCheckData.m_cartErrFlag[i]) AND MasterArmControl.m_masterStatus.m_armState[1] <> MasterArmState_MasterSlave 
								AND MasterArmControl.m_masterStatus.m_armState[2] <> MasterArmState_MasterSlave THEN
		m_cartJoints[i].enable();
	ELSE
		m_cartJoints[i].disable();
	END_IF
	
	// set command position
	m_cartJoints[i].updateCmds(DriverOPMode_Pos,m_cmdJntPos[i],m_cmdJntTrq[i]);
END_FOR
END_METHOD

PROPERTY status : ST_CartStatus
GET
status := m_cartStatus;
END_GET
END_PROPERTY

METHOD PROTECTED updateCmds : BOOL
VAR_INPUT
END_VAR
VAR
	i:INT;
	
END_VAR
IF (m_jntCmdMotionDir[1] <>0 OR m_jntCmdMotionDir[2]<>0 OR m_jntCmdMotionDir[3] <>0 OR m_jntCmdMotionDir[4] <>0) AND m_carInMotion <> 2 THEN
	m_carInMotion := manualAdjust();
ELSIF (m_UIData.m_ergonomicCrl.m_recovErgonEnable OR m_UIData.m_ergonomicCrl.m_cancelRecovErgonEnable) AND m_carInMotion <> 1 THEN
	m_carInMotion := ergonomicAdjust();
ELSE
	m_carInMotion := 0;
END_IF

reachUITargetCheck();
IF m_cmdArrival[1] AND m_cmdArrival[2] AND m_cmdArrival[3] AND m_cmdArrival[4] THEN
	IF m_UIData.m_ergonomicCrl.m_recovErgonEnable THEN
		m_cartStatus.m_cancelErgonAdjustArrival := FALSE;
		m_cartStatus.m_ergonAdjustArrival := TRUE;
	END_IF
	IF m_UIData.m_ergonomicCrl.m_cancelRecovErgonEnable THEN
		m_cartStatus.m_ergonAdjustArrival := FALSE;
		m_cartStatus.m_cancelErgonAdjustArrival := TRUE;
	END_IF
ELSE
	m_cartStatus.m_ergonAdjustArrival := FALSE;
	IF m_UIData.m_ergonomicCrl.m_recovErgonEnable THEN
		m_cartStatus.m_cancelErgonAdjustArrival := FALSE;
	END_IF
END_IF
END_METHOD

METHOD PROTECTED updateIO : BOOL
VAR_INPUT
	i_cartUIData : ST_CartUIData;
END_VAR
VAR
	i:INT;
	idxOffset:INT;
END_VAR
// updata IO signals
m_cartStatus.m_clutchSwitch:= m_clutchIOCheck.check(m_clutchPedalIO);
m_cartStatus.m_endoscopeSwitch := m_endoScopeIOCheck.check(m_endoScopePedalIO);
m_cartStatus.m_surgonReady := m_headInCheck.check(m_surgonHeadInIO);
m_cartStatus.m_armSwitch :=m_armSwitchCheck.check(m_armSwitchIO);
m_UIData := i_cartUIData;

//updata Electrotome control
m_elecKnifeCtrlWord := eleKnifeCtrl(MasterArmControl.m_masterStatus.m_armState , MasterArmControl.m_masterStatus.m_teleSlaveArmIdx , MasterArmControl.m_masterInputDataPool.m_slaveStatus.m_instruStauts );

//updata pedal hover and pedal trigger
m_cartStatus. m_pedalHover[1] := m_electricCutLeftAllow OR m_electricCoagulLeftAllow;
m_cartStatus. m_pedalHover[2] := m_electricCutRightAllow OR m_electricCoagulRightAllow;
IF m_electricCutLeftOn AND m_eleCtrlState = 1 THEN
	m_cartStatus.m_electricKnifePedalTrigger[1] := 1;
ELSIF m_electricCoagulLeftOn AND m_eleCtrlState = 1 THEN
	m_cartStatus.m_electricKnifePedalTrigger[1] := 2;
ELSE
	m_cartStatus.m_electricKnifePedalTrigger[1] := 0;
END_IF

IF m_electricCutRightOn AND m_eleCtrlState = 1 THEN
	m_cartStatus.m_electricKnifePedalTrigger[2] := 1;
ELSIF m_electricCoagulRightOn AND m_eleCtrlState = 1 THEN
	m_cartStatus.m_electricKnifePedalTrigger[2] := 2;
ELSE
	m_cartStatus.m_electricKnifePedalTrigger[2] := 0;
END_IF

//update cart joint control switch
FOR i:=1 TO 4 DO 
	idxOffset:= 2*(i-1);
	IF m_cartJointCtrlIOCheck[1+idxOffset].check(m_cartJointCtrlIO[1+idxOffset]) THEN
		m_jntCmdMotionDir[i]:=1;
	ELSIF  m_cartJointCtrlIOCheck[2+idxOffset].check(m_cartJointCtrlIO[2+idxOffset]) THEN
		m_jntCmdMotionDir[i]:=-1;
	ELSE
		m_jntCmdMotionDir[i]:=0;
	END_IF
END_FOR


// if console is already in motion, only check the currently moving joint
IF m_cartStatus.m_consoleInAdjust THEN
	FOR i:=1 TO 4 DO
		IF NOT(m_cartJoints[i].isEnabled()) THEN
			m_jntCmdMotionDir[i] := 0;
		END_IF
	END_FOR
END_IF


// update joint enable flag
FOR i:= 1 TO 4 DO
	IF m_jntCmdMotionDir[i] <> 0 OR m_UIData.m_ergonomicCrl.m_recovErgonEnable OR m_UIData.m_ergonomicCrl.m_cancelRecovErgonEnable THEN
		m_jntEnableFlag[i] := TRUE;
		m_jntEnableCounts[i]:= LIMIT(0, m_jntEnableCounts[i]+1, m_jntEnableCountsThres);
		m_jntDisableCounts[i]:=m_jntEnableCountsThres;
	ELSE
		m_jntEnableCounts[i]:=0;
		m_jntDisableCounts[i]:= LIMIT(0, m_jntDisableCounts[i]-1, m_jntEnableCountsThres);
		m_jntEnableFlag[i] :=m_jntDisableCounts[i]>0; 
	END_IF
END_FOR

// Do not adjust during master-slave control
IF MasterArmControl.m_masterStatus.m_armState[1] = MasterArmState_MasterSlave OR MasterArmControl.m_masterStatus.m_armState[1] = MasterArmState_Endoscope OR
	MasterArmControl.m_masterStatus.m_armState[2] = MasterArmState_MasterSlave OR MasterArmControl.m_masterStatus.m_armState[2] = MasterArmState_Endoscope  THEN
	m_jntCmdMotionDir := g_zeroVec4i;
END_IF
END_METHOD

METHOD PROTECTED updateStatus : BOOL
VAR_INPUT
END_VAR
VAR
	i:INT;
END_VAR
// update cart joints status
FOR i:=1  TO 4 DO
	m_cartJoints[i].updateStatus();
END_FOR

// get joint data
FOR i:=1 TO 4 DO
	m_curMotorPos[i]:=m_cartJoints[i].motorPos;
	m_curLinkPos[i]:=m_cartJoints[i].linkPos;
	m_curJntPos[i]:=m_cartJoints[i].jntPos;
	m_curJntVel[i]:=m_cartJoints[i].jntVel;
	m_curJntTrq[i]:=m_cartJoints[i].jntTrq;
	m_rawJntCurrent[i]:=m_cartJoints[i].rawCurrent;
	m_filtJntCurrent[i]:=m_cartJoints[i].filtCurrent;
	m_cmdJntCurrent[i]:=m_cartJoints[i].cmdCurrent;
END_FOR 

// transfer monitor angle from link side to motor side
m_curLinkPos[2]:= monitorAngLink2Motor(m_cartJoints[2].linkPos);

// get monitor angle
m_cartStatus.m_monitorAngle:= monitorAngLink2ImagiAxis(m_cartJoints[2].linkPos);

// check if cart in motion
m_cartStatus.m_consoleInAdjust:=FALSE;
FOR i:=1 TO 4 DO
	IF m_cartJoints[i].isEnabled() THEN
		m_cartStatus.m_consoleInAdjust:=TRUE;
		EXIT;
	END_IF
END_FOR

// check if monitor in motion
m_cartStatus.m_monitorInAdjust:=m_cartJoints[2].isEnabled();

// check if cart in manual adjustment
m_cartStatus.m_consoleInManualAdjust := FALSE;
FOR i:=1 TO 4 DO
	IF m_jntCmdMotionDir[i] <> 0 AND m_cartJoints[i].isEnabled() THEN
		m_cartStatus.m_consoleInManualAdjust := TRUE;
		EXIT;
	END_IF
END_FOR
END_METHOD

END_FUNCTION_BLOCK

// ---- FBs_StateControllers/FB_StateCtrlMatching.TcPOU
// Brief: Master Arm Orientation Matching
FUNCTION_BLOCK PUBLIC FB_StateCtrlMatching EXTENDS FB_MasterArmCtrlBase
VAR_INPUT
END_VAR
VAR_OUTPUT
END_VAR
VAR
	// master-slave orientation match threshold
	m_matchAngleThres :LREAL := 2*g_deg2Rad;
	
	m_cmdRotInMonitor :Mat3d;
	
	m_initSolvedJntPos, m_iteSovlvedJntPos :Vec7d;
	m_IKSuccess :BOOL;
	
	m_matchTrajPlanner : FB_TrajMoveJ;
	m_targetJntPos :Vec7d;
	
	m_maxMatchJntVel:Vec7d:=[1.0, 1.0, 1.0, 2*pi, 3*pi, 3*pi, 5*pi];
	m_maxMatchJntAcc:Vec7d:=[1.0, 1.0, 1.0,  8*pi, 12*pi, 12*pi, 20*pi];
	m_maxMatchJntJerk:Vec7d:=[7(100.0)];
	
	m_rotErrAng :LREAL;
	
	
	m_optRes:bool;

END_VAR

// override this function in each exact controller
METHOD PROTECTED calcCmdJntPos : BOOL

VAR_IN_OUT CONSTANT
	i_slaveIdx :INT;
	i_shoulderPose :ST_Frame;
	i_masterArm :FB_MasterArm;
	i_slaveStatus :ST_SlaveStatus;
END_VAR
var 
	i,j : INT;

	mq4,mq5,mq6,mq7:LREAL;
	q4,q5,q6,q7:LREAL;

	rotErr:Mat3d;
	wristRotInJnt3, wristRotInJnt4 :Mat3d;
	rot, invRot :Mat3d;
	cycleNum:INT;
	
	jnt4MoveRange:LREAL;
	jnt5Bias, jnt4MoveScale :LREAL;
	
	cmdJntErr:Vec7d;

END_VAR
IF m_IKSuccess THEN 
	// check if planner is ready
	IF  m_matchTrajPlanner.isGene = FALSE THEN
		RETURN;
	END_IF
	
	// traj plan
	calcCmdJntPos :=m_matchTrajPlanner.evaluate(m_timePeriod, jntPos=> m_cmdJntPos, jntVel=>m_cmdJntVel, jntAcc=> m_cmdJntAcc);
	
	vecSub(m_targetJntPos, m_cmdJntPos, cmdJntErr);
	
	matTranspose(i_masterArm.curCartPose.m_rot, invRot);
	matMultiply(invRot, m_cmdCartPose.m_rot, rotErr);
	rot2AngAxis(rotErr, angle=>m_rotErrAng,axis=>);
	m_isFinished := m_timePeriod > m_matchTrajPlanner.duration AND  norm(cmdJntErr)<g_jntCtrlAngTolHigh and abs(m_rotErrAng)<g_jntCtrlAngTolHigh;
	
	RETURN;
END_IF

// command rotation in monitor
m_cmdRotInMonitor := i_slaveStatus.m_curArmPose[i_slaveIdx].m_rot;

// command rotation in master arm base
matTranspose(i_shoulderPose.m_rot, invRot);
matMultiply(invRot, m_cmdRotInMonitor, m_cmdCartPose.m_rot);
m_cmdCartPose.m_pos:= i_masterArm.curCartPose.m_pos;

// calculate current orientation error
matTranspose(i_masterArm.curCartPose.m_rot, invRot);
matMultiply(invRot, m_cmdCartPose.m_rot, rotErr);
rot2AngAxis(rotErr, angle=>m_rotErrAng,axis=>);

// try IK with optimized posture
rot:=calcJnt3Rotation(m_cmdJntPos[1],m_cmdJntPos[2],m_cmdJntPos[3]);
matTranspose(rot, invRot);
matMultiply(invRot, m_cmdCartPose.m_rot, wristRotInJnt3);
IF 1=i_masterArm.armIdx THEN
	m_IKSuccess := leftWristOptIK(wristRotInJnt3,q4=>q4, q5=>q5, q6=>q6, q7=>q7);
ELSE
	m_IKSuccess := rightWristOptIK(wristRotInJnt3,q4=>q4, q5=>q5, q6=>q6, q7=>q7);
END_IF

// try IK with joint4 at minimal limit
IF NOT m_IKSuccess THEN
	q4:= GVL_ArmJointParameters.g_minJntPos[i_masterArm.armIdx,4];
	
	rot:=calcJnt4Rotation(m_cmdJntPos[1],m_cmdJntPos[2],m_cmdJntPos[3],q4);
	matTranspose(rot, invRot);
	matMultiply(invRot, m_cmdCartPose.m_rot, wristRotInJnt4);
	m_IKSuccess := wristIK(wristRotInJnt4,i_masterArm, q5=>q5, q6=>q6, q7=>q7);
END_IF

// try IK with joint4 at maximum limit
IF NOT m_IKSuccess THEN
	q4:= GVL_ArmJointParameters.g_maxJntPos[i_masterArm.armIdx,4];
	
	rot:=calcJnt4Rotation(m_cmdJntPos[1],m_cmdJntPos[2],m_cmdJntPos[3],q4);
	matTranspose(rot, invRot);
	matMultiply(invRot, m_cmdCartPose.m_rot, wristRotInJnt4);
	m_IKSuccess := wristIK(wristRotInJnt4,i_masterArm, q5=>q5, q6=>q6, q7=>q7);
END_IF

// minimize joint4 move angle
IF m_IKSuccess THEN
	
	// minimize based on join5 posture
	jnt4MoveRange :=  i_masterArm.jnt4LinkToMotor(m_targetJntPos[2],m_targetJntPos[3],q4)-i_masterArm.curJntPos[4];
	jnt5Bias :=  LIMIT (0, ABS(q5-pi), pi/2);
	jnt4MoveRange := jnt4MoveRange * ABS(COS(jnt5Bias));
	
	// minimize based on cartesian error
	IF ABS(m_rotErrAng)< 5.0 * g_deg2Rad THEN
		jnt4MoveRange := 0.0;
	END_IF
	
	mq4:=  i_masterArm.jnt4MotorToLink(m_targetJntPos[2],m_targetJntPos[3],i_masterArm.curJntPos[4] + jnt4MoveRange) ;
	
	rot:=calcJnt4Rotation(m_cmdJntPos[1],m_cmdJntPos[2],m_cmdJntPos[3],mq4);
	matTranspose(rot, invRot);
	matMultiply(invRot, m_cmdCartPose.m_rot, wristRotInJnt4);
	IF wristIK(wristRotInJnt4,i_masterArm, q5=>mq5, q6=>mq6, q7=>mq7) THEN
		q4:=mq4;
		q5:=mq5;
		q6:=mq6;
		q7:=mq7;
	END_IF
END_IF

// traj plan
IF m_IKSuccess THEN 
	m_targetJntPos:=m_cmdJntPos;
	m_targetJntPos[4]:=i_masterArm.jnt4LinkToMotor(m_targetJntPos[2],m_targetJntPos[3],q4);
	m_targetJntPos[5]:=q5;
	m_targetJntPos[6]:=q6;
	
	// roll flip handle
	i_masterArm.flipGripper(rollFlipHandle(i_masterArm.armIdx,i_masterArm.curJntPos[7], q7, o_cmdJntPos7 =>m_targetJntPos[7]));
	
	// no match for rotate joint if instrument is ultrasonic knife
	IF MasterArmControl.m_masterRobot.m_USKnifeRotClutch[i_slaveIdx] THEN
		m_targetJntPos[7] := i_masterArm.curJntPos[7];
	END_IF

	m_matchTrajPlanner.init(m_cmdJntPos,m_targetJntPos,m_maxMatchJntVel,m_maxMatchJntAcc,m_maxMatchJntJerk);
	m_timePeriod :=0;
END_IF
END_METHOD

// calculate joint3 rotation in arm coordinate
(*armDH=[   0      0   q1      d1;
            -deg90  0   q2      0;
            0       a3  q3      0];*)
METHOD PROTECTED calcJnt3Rotation : Mat3d
VAR_INPUT CONSTANT
	q1:LREAL;
	q2:LREAL;
	q3:LREAL;
END_VAR

VAR
	c1,c2,c3,s1,s2,s3,c23,s23 :LREAL;
END_VAR
// !Convert active joint position to DH model for kinematic calculation
q3:=q3-q2;  //q3=q8-q2

c1:=COS(q1);
c2:=COS(q2);
c3:=COS(q3);

s1:=SIN(q1);
s2:=SIN(q2);
s3:=SIN(q3);

c23:=COS(q2+q3);
s23:=SIN(q2+q3);

calcJnt3Rotation[1,1]:= c23*c1;
calcJnt3Rotation[2,1]:= c23*s1;
calcJnt3Rotation[3,1]:= -s23;

calcJnt3Rotation[1,2]:= -s23*c1;
calcJnt3Rotation[2,2]:= -s23*s1;
calcJnt3Rotation[3,2]:= -c23;

calcJnt3Rotation[1,3]:= -s1;
calcJnt3Rotation[2,3]:= c1;
calcJnt3Rotation[3,3]:=0;
END_METHOD

// calculate joint3 rotation in arm coordinate
(*[   0      0   q1      d1;
	-deg90  0   q2      0;
	0       a3  q3      0;
	 -deg90  a4  q4      d4]
*)
METHOD PROTECTED calcJnt4Rotation : Mat3d
VAR_INPUT
	q1 :LREAL;
	q2 :LREAL;
	q3 :LREAL;
	q4 :LREAL;// already at the link side
END_VAR

VAR
	c1,c2,c3,c4, s1,s2,s3,s4,c23,s23 :LREAL;
END_VAR
// !Convert active joint position to DH model for kinematic calculation
//q4:=q4+q3-q2-pi/2;//q4DH=q4motor+q8-q2-90;  
q3:=q3-q2;  //q3=q8-q2

c1:=COS(q1);
c2:=COS(q2);
c3:=COS(q3);
c4:=COS(q4);

s1:=SIN(q1);
s2:=SIN(q2);
s3:=SIN(q3);
s4:=SIN(q4);

c23:=COS(q2+q3);
s23:=SIN(q2+q3);

calcJnt4Rotation[1,1]:= s1*s4 + c4*c1*c23;
calcJnt4Rotation[2,1]:= - c1*s4 + c4*s1*c23;
calcJnt4Rotation[3,1]:= -s23*c4;

calcJnt4Rotation[1,2]:= c4*s1 - s4*c1*c23;
calcJnt4Rotation[2,2]:= -s4*s1*c23 - c1*c4;
calcJnt4Rotation[3,2]:=   s23*s4;

calcJnt4Rotation[1,3]:= -s23*c1;
calcJnt4Rotation[2,3]:= -s23*s1;
calcJnt4Rotation[3,3]:=-c23;
END_METHOD

PROPERTY IKSuccess : BOOL
GET
IKSuccess := m_IKSuccess;
END_GET
END_PROPERTY

METHOD PUBLIC init : BOOL
VAR_IN_OUT CONSTANT
	i_masterArm	:FB_MasterArm;
END_VAR
VAR_IN_OUT 
	r_masterArmCtrlCmd :ST_ArmCtrlCmds;
END_VAR
// check if to hold the command joint position unchanged
m_holdLastCmds := checkToHoldLastCmds(i_masterArm);

// init
SUPER^.Init(i_masterArm,r_masterArmCtrlCmd);

m_jntOPMode[4]:=DriverOPMode_PosTrq;
m_jntOPMode[5]:=DriverOPMode_PosTrq;
m_jntOPMode[6]:=DriverOPMode_PosTrq;
m_jntOPMode[7]:=DriverOPMode_PosTrq;

m_IKSuccess:=FALSE;
m_targetJntPos:=m_cmdJntPos;

// update commands to arm
copyCmds(r_masterArmCtrlCmd);
END_METHOD

// calculate command wrist joint position with an optimized posture
(*wristDH=[   -deg90  a4  q4      d4;
            deg90   0   q5      0;
            -deg90  0   q6      0;
            deg90   0   q7      0];*)
// set q6 = -pi/2 for desired posture
(* wristRot = 
[ COS(q7)*SIN(q4) - COS(q4)*SIN(q5)*SIN(q7), - SIN(q4)*SIN(q7) - COS(q4)*COS(q7)*SIN(q5), -COS(q4)*COS(q5)]
[                           cos(q5)*sin(q7),                             cos(q5)*cos(q7),         -sin(q5)]
[ cos(q4)*cos(q7) + sin(q4)*sin(q5)*sin(q7),   cos(q7)*sin(q4)*sin(q5) - cos(q4)*sin(q7),  cos(q5)*sin(q4)]
*)
METHOD PROTECTED leftWristOptIK : BOOL
VAR_IN_OUT CONSTANT
	i_cmdRot :Mat3d;
END_VAR
VAR_OUTPUT
	q4 :LREAL;
	q5 :LREAL;
	q6 :LREAL;
	q7 :LREAL;
END_VAR

VAR
	q51,q52 :LREAL;
	s4,c4,s5,c5,s7,c7:LREAL;
	q4UnreachPosMin: LREAL :=-pi/2;
	q4UnreachPosMax: LREAL :=45*g_deg2Rad;
	
END_VAR
q6:=-PI/2;
// q5 = [pi-135deg, pi+135deg]
q5 := ASIN(-i_cmdRot[2,3]);
q5:= PI-q5;

// q5=3pi/2 or q5=pi/2
IF ABS(q5-3*PI/2)<g_smallAng OR ABS(q5-PI/2)<g_smallAng THEN
	q4:= -pi;
	s7:= -i_cmdRot[1,1]/(COS(q4)*SIN(q5));
	c7:= i_cmdRot[3,1]/COS(q4);
	q7:=atan2(s7,c7);
	leftWristOptIK:=TRUE;
	RETURN;
END_IF

// solution one 
c5 :=COS(q5);
s7:=i_cmdRot[2,1]/c5;
c7:= i_cmdRot[2,2]/c5;
q7:=atan2(s7,c7);

//q4=[-pi/2-225deg, -pi/2]
c4 := -i_cmdRot[1,3]/c5;
s4:= i_cmdRot[3,3]/c5;
q4:=atan2(s4,c4);
IF q4> GVL_ArmJointParameters.g_minJntPos[1,4] AND q4<GVL_ArmJointParameters.g_maxJntPos[1,4] THEN
	leftWristOptIK:=TRUE;
	RETURN;
ELSIF q4> GVL_ArmJointParameters.g_maxJntPos[1,4] AND q4-2*pi> GVL_ArmJointParameters.g_minJntPos[1,4] THEN
	q4:=q4-2*PI;
	leftWristOptIK:=TRUE;
	RETURN;
END_IF

// solution2
IF q5 > pi THEN
	q5 := 3*PI-q5;
ELSE
	q5:= pi-q5;
END_IF
IF q5 > GVL_ArmJointParameters.g_maxJntPos[1,5] OR q5<GVL_ArmJointParameters.g_minJntPos[1,5] THEN
	leftWristOptIK:=FALSE;
	RETURN;
END_IF

c5 :=COS(q5);
s7:=i_cmdRot[2,1]/c5;
c7:= i_cmdRot[2,2]/c5;
q7:=atan2(s7,c7);

c4 := -i_cmdRot[1,3]/c5;
s4:= i_cmdRot[3,3]/c5;
q4:=atan2(s4,c4);
IF q4> GVL_ArmJointParameters.g_minJntPos[1,4] AND q4<GVL_ArmJointParameters.g_maxJntPos[1,4] THEN
	leftWristOptIK:=TRUE;
	RETURN;
ELSIF q4> GVL_ArmJointParameters.g_maxJntPos[1,4] AND q4-2*pi< GVL_ArmJointParameters.g_minJntPos[1,4] THEN
	q4:=q4-2*PI;
	leftWristOptIK:=TRUE;
	RETURN;
END_IF
END_METHOD

// calculate command wrist joint position with an optimized posture
(*wristDH=[   -deg90  a4  q4      d4;
            deg90   0   q5      0;
            -deg90  0   q6      0;
            deg90   0   q7      0];*)
// set q6 = pi/2 for desired posture
(* wristRot = 
[ - cos(q7)*sin(q4) - cos(q4)*sin(q5)*sin(q7), sin(q4)*sin(q7) - cos(q4)*cos(q7)*sin(q5),  cos(q4)*cos(q5)]
[                             cos(q5)*sin(q7),                           cos(q5)*cos(q7),          sin(q5)]
[   sin(q4)*sin(q5)*sin(q7) - cos(q4)*cos(q7), cos(q4)*sin(q7) + cos(q7)*sin(q4)*sin(q5), -cos(q5)*sin(q4)]
 
*)
METHOD PROTECTED rightWristOptIK : BOOL
VAR_IN_OUT CONSTANT
	i_cmdRot :Mat3d;
END_VAR
VAR_OUTPUT
	q4 :LREAL;
	q5 :LREAL;
	q6 :LREAL;
	q7 :LREAL;
END_VAR

VAR
	q51,q52 :LREAL;
	s4,c4,s5,c5,s7,c7:LREAL;
	q4UnreachPosMin: LREAL :=-pi/2;
	q4UnreachPosMax: LREAL :=45*g_deg2Rad;
	
END_VAR
q6:=PI/2;
// q5 = [pi-135deg, pi+135deg]
q5 := ASIN(i_cmdRot[2,3]);
q5:= PI-q5;

// q5=3pi/2 or q5=pi/2
IF ABS(q5-3*PI/2)<g_smallAng OR ABS(q5-PI/2)<g_smallAng THEN
	q4:= 0;
	s7:= -i_cmdRot[1,1]/(COS(q4)*SIN(q5));
	c7:= -i_cmdRot[3,1]/COS(q4);
	q7:=atan2(s7,c7);
	rightWristOptIK:=TRUE;
	RETURN;
END_IF

// solution one 
c5 :=COS(q5);
s7:=i_cmdRot[2,1]/c5;
c7:= i_cmdRot[2,2]/c5;
q7:=atan2(s7,c7);

//q4=[-pi/2, -pi/2+225deg]
c4 := i_cmdRot[1,3]/c5;
s4:= -i_cmdRot[3,3]/c5;
q4:=atan2(s4,c4);
IF q4> GVL_ArmJointParameters.g_minJntPos[2,4] AND q4<GVL_ArmJointParameters.g_maxJntPos[2,4] THEN
	rightWristOptIK:=TRUE;
	RETURN;
END_IF

// solution2
IF q5 > pi THEN
	q5 := 3*PI-q5;
ELSE
	q5:= pi-q5;
END_IF
IF q5 > GVL_ArmJointParameters.g_maxJntPos[1,5] OR q5<GVL_ArmJointParameters.g_minJntPos[1,5] THEN
	rightWristOptIK:=FALSE;
	RETURN;
END_IF

c5 :=COS(q5);
s7:=i_cmdRot[2,1]/c5;
c7:= i_cmdRot[2,2]/c5;
q7:=atan2(s7,c7);

//q4=[-pi/2, -pi/2+225deg]
c4 := i_cmdRot[1,3]/c5;
s4:= -i_cmdRot[3,3]/c5;
q4:=atan2(s4,c4);
IF q4> GVL_ArmJointParameters.g_minJntPos[2,4] AND q4<GVL_ArmJointParameters.g_maxJntPos[2,4] THEN
	rightWristOptIK:=TRUE;
	RETURN;
END_IF
END_METHOD

METHOD PROTECTED rollFlipHandle : BOOL
VAR_INPUT
	i_armIdx:INT;
	i_curJntPos7 :LREAL;
	i_initCmdJntPos7 :LREAL;
END_VAR
VAR_OUTPUT
	o_cmdJntPos7 :LREAL;
END_VAR

VAR
	solFeasible1,solFeasible2 :BOOL;
	solIdx :INT:=0;
	halfcycleNum1, halfcycleNum2:INT;
	solution1, solution2 :LREAL;
END_VAR
// this part is used to drive gripper back near center, in case that gripper roll is stuck near limit
// TODO: remove after gripper roll has infinite motion range
//IF NOT (MasterArmControl.m_masterInputDataPool.m_cartStatus.m_surgonReady) THEN
//	o_cmdJntPos7:=i_initCmdJntPos7;
//	rollFlipHandle:=FALSE;
//	RETURN;
//END_IF

// handle multiple cycles of joint7
// find the first solution within pi from current position
halfcycleNum1 := LREAL_TO_INT((i_curJntPos7 - i_initCmdJntPos7)/pi);
solution1 := halfcycleNum1 * pi + i_initCmdJntPos7;

// solution2
IF solution1 > i_curJntPos7 THEN
	solution2 := solution1 - PI;
	halfcycleNum2 := halfcycleNum1 - 1;
ELSE
	solution2 := solution1 + PI;
	halfcycleNum2 := halfcycleNum1 + 1;
END_IF

//choose the solution which is closer to current q7 which can achive orientation match with a max pi/2 degree
// NOTE: There maybe risk this joint7 is stuck at limit, which can be solved after joint7 has infinite rotation angle,
solFeasible1:=solution1> GVL_ArmJointParameters.g_minJntPos[i_armIdx,7] AND solution1< GVL_ArmJointParameters.g_maxJntPos[i_armIdx,7];
solFeasible2:=solution2> GVL_ArmJointParameters.g_minJntPos[i_armIdx,7] AND solution2< GVL_ArmJointParameters.g_maxJntPos[i_armIdx,7];
IF solFeasible1 AND solFeasible2 THEN
	IF ABS(solution1-i_curJntPos7) < ABS(solution2-i_curJntPos7)  THEN
		solIdx:=1;
	ELSE
		solIdx:=2;
	END_IF
ELSIF solFeasible1 AND NOT(solFeasible2) THEN
	solIdx:=1;
ELSIF solFeasible2 AND NOT(solFeasible1) THEN
	solIdx:=2;
ELSE
	solIdx:=0;
END_IF

IF solIdx = 1 THEN
	o_cmdJntPos7 := solution1;
	rollFlipHandle:= ((ABS(halfcycleNum1) MOD 2) = 1);
ELSIF solIdx =2 THEN
	o_cmdJntPos7 := solution2;
	rollFlipHandle:= ((ABS(halfcycleNum2) MOD 2) = 1);
ELSE
	o_cmdJntPos7:=i_initCmdJntPos7;
	rollFlipHandle:=FALSE;
END_IF
END_METHOD

// calculate position of joint 5/6/7 
(*wristDH=[   deg90   0   q5      0;
            -deg90  0   q6      0;
            deg90   0   q7      0];*)
(* wristRot = 
[ cos(q5)*cos(q6)*cos(q7) - sin(q5)*sin(q7), - cos(q7)*sin(q5) - cos(q5)*cos(q6)*sin(q7), cos(q5)*sin(q6)]
[                           cos(q7)*sin(q6),                            -sin(q6)*sin(q7),        -cos(q6)]
[ cos(q5)*sin(q7) + cos(q6)*cos(q7)*sin(q5),   cos(q5)*cos(q7) - cos(q6)*sin(q5)*sin(q7), sin(q5)*sin(q6)]
*)
METHOD PROTECTED wristIK : BOOL
VAR_IN_OUT CONSTANT
	i_cmdRot :Mat3d;
	i_masterArm :FB_MasterArm;
END_VAR

VAR_OUTPUT
	q5:	LREAL;
	q6:	LREAL;
	q7:	LREAL;
END_VAR

VAR
	invRot :Mat3d;
	jnt4Rotation :Mat3d;
	s5, s7, c5, c7:LREAL;
END_VAR
// calculate wrist joint position
// q6=[-pi/2-45deg, -pi/2+45deg]
IF 1 = i_masterArm.armIdx THEN
	q6:= -ACOS(-i_cmdRot[2,3]);
// q6=[pi/2-45deg, pi/2+45deg]
ELSE
	q6:= ACOS(-i_cmdRot[2,3]);
END_IF

IF q6>GVL_ArmJointParameters.g_maxJntPos[i_masterArm.armIdx, 6] OR q6< GVL_ArmJointParameters.g_minJntPos[i_masterArm.armIdx, 6] THEN
	wristIK:=FALSE;
	RETURN;
END_IF

// q5 = [pi-135deg, pi+135deg]
c5 := i_cmdRot[1,3]/SIN(q6);
s5 := i_cmdRot[3,3]/SIN(q6);
q5:=atan2(s5,c5);
IF q5<GVL_ArmJointParameters.g_minJntPos[1,5] THEN
	q5:=q5+2*PI;
END_IF
IF q5>GVL_ArmJointParameters.g_maxJntPos[1,5]THEN
	wristIK:=FALSE;
	RETURN;
END_IF
c7 := i_cmdRot[2,1]/SIN(q6);
s7 := -i_cmdRot[2,2]/SIN(q6);
q7:=atan2(s7,c7);
wristIK:=true;
END_METHOD

END_FUNCTION_BLOCK

// ---- FBs_Robots/FB_MasterRobot.TcPOU
FUNCTION_BLOCK FB_MasterRobot
VAR
	// flag if slave are connected
	m_slaveOnLine :BOOL :=FALSE;
	m_slaveOnLineCheck :FB_slaveConnectionCheck;
	
	// master-slave motion scale
	m_motionScale :LREAL;
	
	// monitor angle
	m_monitorAngle :LREAL;
	
	// master arm base pose(shoulder pose) in monitor coordinate
	m_shoulderPoseInMonitor :ARRAY[1..2] OF ST_Frame;
	
	// master arms, responsible for arm kinematic and control
	m_masterArms :ARRAY[1..g_mArmNum] OF FB_MasterArm;
	
	// arm state
	m_masterArmState:ARRAY[1..g_mArmNum] OF E_masterArmState:=[E_masterArmState.MasterArmState_Init,E_masterArmState.MasterArmState_Error];
	m_lastMasterArmState:ARRAY[1..g_mArmNum] OF E_masterArmState:=[E_masterArmState.MasterArmState_Init,E_masterArmState.MasterArmState_Error];
	m_nextMasterArmState:ARRAY[1..g_mArmNum] OF E_masterArmState:=[E_masterArmState.MasterArmState_Init,E_masterArmState.MasterArmState_Error];
	
	// index(1 to 4) of slave arm which is tele-linked to master arm
	m_teleSlaveArmIdx:ARRAY[1..g_mArmNum] OF E_MatchedSlaveArmIdx:=[MatchedSlaveArmIdx_NULL, MatchedSlaveArmIdx_null];
	m_matchedMasterArmIdx :ST_MatchedMasterArmIdx;
	m_instruArmState:ARRAY [1..g_mArmNum] OF E_SlaveArmState:=[SlaveArmState_Error, SlaveArmState_Error];
	m_scopeArmState :E_SlaveArmState := SlaveArmState_Error;
	m_scopeArmIndex : E_MatchedSlaveArmIdx :=MatchedSlaveArmIdx_null;
	
	// flag if tele-manipulated slave arm is switched
	m_armSwitchFlag :ARRAY[1..2] OF BOOL := [2(FALSE)];
	
	//master arm selfcheck finshed flag
	m_armSelfCheckFinshedFlag :ARRAY [1..2] OF BOOL;
	
	// flag to enter master-slave control, triggerd by pinching the gripper twice in on second
	m_MSCtrlTriggerFlag :ARRAY[1..g_mArmNum] OF BOOL:=[FALSE, FALSE];
	m_MSCtrlTriggerCheck :ARRAY[1..g_mArmNum] OF FB_MSCtrlTriggerCheck;
	
	// all arm controller instance 
	m_armCtrlFactory :ARRAY[1..g_mArmNum,1..MasterArmState_totalNum] OF I_MasterArmCtrl;
	m_armError :ARRAY[1..g_mArmNum] OF FB_StateCtrlError;
	m_armInit :ARRAY[1..g_mArmNum] OF FB_StateCtrlInit;
	m_armHome :ARRAY[1..g_mArmNum] OF FB_StateCtrlHome;
	m_armStandBy :ARRAY[1..g_mArmNum] OF FB_StateCtrlStandBy;
	m_armMatching :ARRAY[1..g_mArmNum] OF FB_StateCtrlMatching;
	m_armReady :ARRAY[1..g_mArmNum] OF FB_StateCtrlReady;
	m_armMasterSlave :ARRAY[1..g_mArmNum] OF FB_StateCtrlMasterSlave;
	m_armClutch :ARRAY[1..g_mArmNum] OF FB_StateCtrlClutch;
	m_armEndoscope :ARRAY[1..g_mArmNum] OF FB_StateCtrlEndoscope;
	m_armCart :ARRAY[1..g_mArmNum] OF FB_StateCtrlCart;
	m_armGravityCali :ARRAY[1..g_mArmNum] OF FB_StateCtrlGraCali;
	m_armTest :ARRAY[1..g_mArmNum] OF FB_StateCtrlTest;
	m_armDisable :ARRAY[1..g_mArmNum] OF FB_StateCtrlDisable;
	m_armPerformance :ARRAY[1..g_mArmNum] OF FB_StateCtrlPerformance;
	
	// specialized endoscope controller
	m_scopeCtrl :FB_EndoscopeController;
	
	// arm controller interface
	m_armCtrl :ARRAY[1..g_mArmNum] OF I_MasterArmCtrl;
	m_armCtrlCmds :ARRAY[1..g_mArmNum] OF ST_ArmCtrlCmds;
	
	// ultrasonic knife rotation clutch flag
	m_USKnifeRotClutch :ARRAY[1..g_sArmNum] OF BOOL := [4(FALSE)];

END_VAR

 METHOD PROTECTED checkTeleSlaveArmIdx : BOOL
VAR_IN_OUT CONSTANT
	i_masterInputDataPool:ST_MasterInputDataPool;
END_VAR
VAR_STAT
	m_armSwitchR : R_TRIG;
	m_armSwitch : BOOL;
	nextTeleSlaveArmIdx:ARRAY[1..g_mArmNum] OF E_MatchedSlaveArmIdx;
END_VAR
nextTeleSlaveArmIdx:=m_teleSlaveArmIdx;
m_armSwitchR(CLK:= i_masterInputDataPool.m_cartStatus.m_armSwitch, Q=> m_armSwitch);
IF m_armSwitch THEN
	m_matchedMasterArmIdx.left1ArmIdx := GVL_interactUI.g_armDistributionInfo.m_leftMappingSlaveArm[1];
	m_matchedMasterArmIdx.left2ArmIdx := GVL_interactUI.g_armDistributionInfo.m_leftMappingSlaveArm[2];
	m_matchedMasterArmIdx.right1ArmIdx := GVL_interactUI.g_armDistributionInfo.m_rightMappingSlaveArm[1];
	m_matchedMasterArmIdx.right2ArmIdx := GVL_interactUI.g_armDistributionInfo.m_rightMappingSlaveArm[2];
END_IF


IF m_matchedMasterArmIdx.left1ArmIdx <=0 OR m_matchedMasterArmIdx.left2ArmIdx <=0 OR m_matchedMasterArmIdx.right1ArmIdx <=0 OR m_matchedMasterArmIdx.right2ArmIdx <=0 THEN
	RETURN;
END_IF

// switch tele-controlled arm index when arm is disenabled
IF i_masterInputDataPool.m_slaveStatus.m_armState[m_matchedMasterArmIdx.left1ArmIdx] = SlaveArmState_Disable THEN
	nextTeleSlaveArmIdx[1]:= m_matchedMasterArmIdx.left2ArmIdx;
ELSIF i_masterInputDataPool.m_slaveStatus.m_armState[m_matchedMasterArmIdx.left2ArmIdx] = SlaveArmState_Disable THEN
	nextTeleSlaveArmIdx[1]:= m_matchedMasterArmIdx.left1ArmIdx;
ELSIF i_masterInputDataPool.m_slaveStatus.m_armState[m_matchedMasterArmIdx.right1ArmIdx] = SlaveArmState_Disable THEN
	nextTeleSlaveArmIdx[2]:= m_matchedMasterArmIdx.right2ArmIdx;
ELSIF i_masterInputDataPool.m_slaveStatus.m_armState[m_matchedMasterArmIdx.right2ArmIdx] = SlaveArmState_Disable THEN
	nextTeleSlaveArmIdx[2]:= m_matchedMasterArmIdx.right1ArmIdx;
END_IF


// switch tele-controlled arm index when endoscope is mounted
IF m_scopeArmIndex = m_matchedMasterArmIdx.left1ArmIdx OR m_scopeArmIndex = m_matchedMasterArmIdx.left2ArmIdx THEN
	// left arm
	IF m_scopeArmIndex = m_matchedMasterArmIdx.left1ArmIdx THEN
		nextTeleSlaveArmIdx[1] := m_matchedMasterArmIdx.left2ArmIdx;
	ELSE
		nextTeleSlaveArmIdx[1] := m_matchedMasterArmIdx.left1ArmIdx;
	END_IF
	
	// right arm
	// switch tele-controlled arm index when arm switch is triggerd
	IF m_armSwitch THEN
		IF m_teleSlaveArmIdx[2] = m_matchedMasterArmIdx.right1ArmIdx AND i_masterInputDataPool.m_slaveStatus.m_armState[m_matchedMasterArmIdx.right2ArmIdx]=SlaveArmState_InstruReady THEN
			nextTeleSlaveArmIdx[2] := m_matchedMasterArmIdx.right2ArmIdx;
		ELSIF 
			m_teleSlaveArmIdx[2]=m_matchedMasterArmIdx.right2ArmIdx AND i_masterInputDataPool.m_slaveStatus.m_armState[m_matchedMasterArmIdx.right1ArmIdx]=SlaveArmState_InstruReady THEN
			nextTeleSlaveArmIdx[2] := m_matchedMasterArmIdx.right1ArmIdx;
		ELSE
			IF  i_masterInputDataPool.m_slaveStatus.m_armState[m_matchedMasterArmIdx.right1ArmIdx]=SlaveArmState_InstruReady THEN
				nextTeleSlaveArmIdx[2] := m_matchedMasterArmIdx.right1ArmIdx;
			ELSIF i_masterInputDataPool.m_slaveStatus.m_armState[m_matchedMasterArmIdx.right2ArmIdx]=SlaveArmState_InstruReady THEN
				nextTeleSlaveArmIdx[2] := m_matchedMasterArmIdx.right2ArmIdx;
			ELSE
				nextTeleSlaveArmIdx[2] := m_matchedMasterArmIdx.right1ArmIdx;
			END_IF
			
		END_IF
	END_IF

